  (*From Machine*)
  bI_DeviceOnline            : BOOL;	(*Check link to device*)
  bI_Sensor_pA               : BOOL;	(*Physical sensor feedback for pA Position *)
  bI_Sensor_pB               : BOOL;	(*Physical sensor feedback for pB Position *)
  bI_SystemReady             : BOOL;	(*General ready flag*)
  bI_MovementAllowed         : BOOL;	(*No collision danger*)
  bI_HomingAllowed           : BOOL;	(*Homing allowed*)
  bI_SafetyOk                : BOOL;	(*Safety ok for movement*)
  bI_AbortCleaning           : BOOL;	(*Abort cleaning, drive to pA*)

  (*Commands from Cleaning Process Controller*)
  sI_CleanDevCmd             : ST_CLEANING_DEV_CMD;	(*Initialize operation*)

  (*From User*)
  sI_ManualCommands          : ST_MANUAL_CMD;
  bI_AckFault                : BOOL;	(* Acknowledge errors*)
  bI_Enable                  : BOOL;	(* Enable PrintUnit axis*)
  fI_Position_p1             : REAL;
  fI_Position_p2             : REAL;
  fI_Position_A              : REAL;
  fI_Position_B              : REAL;
  fI_PositionTolerance       : REAL := 0.001;
  fI_SetPositionValue        : REAL := 0.0;    (*Set position value [m]*)
  sI_SpeedDef_Y              : ST_SPEEDS;	(*Speed defs*)
  bI_ShinyMode               : BOOL;	(*Cleaning option*)
  bI_EnableBinClean          : BOOL := TRUE;

  (*From Motor Controller*)
  eI_ELmodule_State          : EN_EL7201_STATE;	(*Feedback from Axis*)
  bI_MoveDone                : BOOL;
  fI_CurrentPosition         : REAL;

  pC_MsgInterface            : POINTER TO ST_ADS_MSG_IF;
  iC_BlockId                 : INT;
END_VAR

VAR_OUTPUT
  (*To Cleaning Head*)
  bO_EnableClnHead           : BOOL;
  bO_EnableVacuum            : BOOL;

  (*To Motor Controller*)
  fO_TargetPosition          : REAL;	(*Target position for axis*)
  fO_SpeedLimit              : REAL;	(*Speed limit for axis*)
  bO_MoveEnable              : BOOL;	(*Move enable for axis*)
  bO_RegActive               : BOOL;	(*Close control loop for axis*)
  bO_FaultReset              : BOOL;	(*Fault reset for axis*)
  bO_SetPosition             : BOOL; (*Reset Encoder*)
  bO_PositionUnknown         : BOOL; (*Position of axis is unknown*)

  (*To machine/user*)
  sO_CleanDevStatus          : ST_CLEANING_DEV_STATUS;	(*Initialize operation*)
  sO_ClnHead_Mvt_Status      : ST_CH_MVT_STATUS;
  bO_CleanAborted            : BOOL;  (*Cleaning aborted*)
END_VAR

VAR
  cL_State                   : BYTE;	(*State type*)
  bL_CleaningActive          : BOOL;
  bL_AfterCleaning           : BOOL := FALSE;
  bL_AxisReady               : BOOL;
  bL_CleanActive             : BOOL;
  bL_MoveAReq                : BOOL;
  bL_MoveBReq                : BOOL;
  bL_MoveDone                : BOOL;
  bL_SafeRunningCondition    : BOOL;
  bL_SafeMoveNeg             : BOOL;
  bL_SafeMovePos             : BOOL;
  bL_Ref_Known               : BOOL := FALSE;
  bL_MoveStarted             : BOOL := FALSE;
  bL_MoveStartRequested      : BOOL := FALSE;

  bL_InPosA                  : BOOL;
  bL_InPosB                  : BOOL;

  wL_ErrorCode               : WORD;

  bL_MotionActive            : BOOL;

  tL_TimerSurv               : TON;			(* Timer for Motorization check *)
  tL_TimerSensor             : TON;			(* Timer for Sensor check *)
  bL_memRefSensor            : BOOL;
  bL_memAck                  : BOOL;
  bL_mem_MotionActive        : BOOL;
  bL_mem_MoveEnable          : BOOL;
  bL_FirstRun                : BOOL := TRUE;
  tL_TonMoveAReq             : TON;			(* Timer for moving back to A *)

  (*Messaging*)
  fB_MsgQueue                : FB_MSG_QUEUE;
  fB_MsgHandler              : FB_MSG_HANDLER;
  sL_MsgConfig               : ST_MSG_CONFIG;
  fB_Msg                     : ARRAY [1..iC_NUM_MSG] OF FB_MESSAGE;
END_VAR

VAR CONSTANT
	(*State*)
  cL_IDLE_A                  : BYTE := 0;										(*Idle-State @ Start*)
  cL_MOVE_P1                 : BYTE := 10;										(*Move to Position where Cleaning starts*)
  cL_ENABLE_CLEAN            : BYTE := 20;										(*Enable Cleaning System*)
  cL_MOVE_P2                 : BYTE := 30;										(*Move to Position where Cleaning stops*)
  cL_DISABLE_CLEAN           : BYTE := 40;										(*Disable Cleaning System*)
  cL_MOVE_A                  : BYTE := 50;										(*Move to start*)
  cL_MOVE_A_CLEANBIN         : BYTE := 51;										(*Move to start with cleaning the bin*)
  cL_MOVE_B                  : BYTE := 60;										(*Move to end*)
  cL_IDLE_B                  : BYTE := 70;										(*Idle-State @ Stop*)
  cL_UNKNOWN                 : BYTE := 80;										(*Position unknown*)

  iC_NUM_MSG                 : INT  := 1;
END_VAR

tL_TimerSurv.PT := T#3s;
tL_TimerSurv();
tL_TimerSensor.PT := T#105s	;	(* 1meter at 10mm*)
tL_TimerSensor();

IF bL_FirstRun THEN
	bL_FirstRun     := FALSE;
	bL_memRefSensor := bI_Sensor_pA;
END_IF;

(*----------------------------------------------------------------------------------------------------------------------------------------------- *)
(*Running Conditions  For Cleaning Head  *)
(*----------------------------------------------------------------------------------------------------------------------------------------------- *)
IF bI_SystemReady AND bI_DeviceOnline AND bI_MovementAllowed AND bI_SafetyOk AND (wL_ErrorCode = 0 OR wL_ErrorCode.5)THEN	(*Dont check limit switch here*)
	bL_SafeRunningCondition := TRUE;
ELSE
	bL_SafeRunningCondition := FALSE;
END_IF;

bL_SafeMoveNeg := bL_SafeRunningCondition AND NOT bI_Sensor_pA AND bI_MovementAllowed;
bL_SafeMovePos := bL_SafeRunningCondition AND NOT bI_Sensor_pB AND bI_MovementAllowed;

IF NOT bI_DeviceOnline THEN
	bL_Ref_Known := FALSE;				(*Reset Reference when link to device is lost, e.g. when machine power off*)
END_IF;

(*----------------------------------------------------------------------------------------------------------------------------------------------- *)
(*Position detection*)
(*----------------------------------------------------------------------------------------------------------------------------------------------- *)

IF     (fI_CurrentPosition >= (fI_Position_A - fI_PositionTolerance)
   AND  fI_CurrentPosition <= (fI_Position_A + fI_PositionTolerance)) OR bI_Sensor_pA
THEN
	bL_InPosA := TRUE;
	bL_InPosB := FALSE;
ELSIF  fI_CurrentPosition >= (fI_Position_B - fI_PositionTolerance)
   AND fI_CurrentPosition <= (fI_Position_B + fI_PositionTolerance)
THEN
	bL_InPosA := FALSE;
	bL_InPosB := TRUE;
ELSE
	bL_InPosA := FALSE;
	bL_InPosB := FALSE;
END_IF;


(*----------------------------------------------------------------------------------------------------------------------------------------------- *)
(* Motion Control For the Cleaning Head 																																																					*)
(*----------------------------------------------------------------------------------------------------------------------------------------------- *)

(*----------------------------------------------------------------------------------------------------------------------------------------------- *)
(*------------------------------------------- Motion Control For the Cleaning Unit   ------------------------------------------------------------ *)
(*----------------------------------------------------------------------------------------------------------------------------------------------- *)
IF NOT bL_Ref_Known THEN	(* if the Y axis hasn't been initialized with Ref Sensor*)
	bL_AxisReady := FALSE;

	IF bI_Sensor_pA AND NOT bL_memRefSensor AND NOT bL_Ref_Known THEN
		bL_Ref_Known    := TRUE;											(* When the sensor is activated, Save the correction value*)
		bL_MotionActive := FALSE;
		bO_SetPosition  := TRUE;											(*Initialize position to preset value*)
		bL_AxisReady    := TRUE;

		fO_TargetPosition := fI_SetPositionValue;
	ELSE
		IF bI_Sensor_pA AND bL_memRefSensor THEN
			fO_TargetPosition := fI_CurrentPosition + 0.01;            (*@@@@CONST, change to JOG_NEGATIVE*)
			fO_SpeedLimit     := sI_SpeedDef_Y.fP_ServiceSpeed;        (* Start backward motion, the motor will run until Ref Sensor is ON*)
			bL_MotionActive   := bI_HomingAllowed;
			bO_SetPosition    := FALSE;
		ELSE
			fO_TargetPosition := -100.0;                               (*@@@@CONST, change to JOG_NEGATIVE*)
			fO_SpeedLimit     := sI_SpeedDef_Y.fP_ServiceSpeed * 0.1;  (* Start backward motion, the motor will run until Ref Sensor is ON*)
			bL_MotionActive   := bI_HomingAllowed;
			bO_SetPosition    := FALSE;
		END_IF;
    (*Security check if sensor malfunction:*)
    (*The CH tries to leave the sensor and drives to side B.*)
    (*If sensor malfunction the axis drives only to the end and stops there.*)
    IF (fO_TargetPosition >= fI_Position_B) THEN
      bL_Ref_Known    := FALSE;
      bL_MotionActive := FALSE;
      bO_SetPosition  := FALSE;
      bL_AxisReady    := FALSE;
		END_IF
	END_IF;
ELSE	(* If the axis has been initialized *)
	IF sI_CleanDevCmd.bService THEN
		ServiceMode();
	ELSE
		ProductionMode();
	END_IF;
END_IF;
bL_memRefSensor := bI_Sensor_pA;				(* Memorization of the Ref sensor state for edge detection*)
bO_RegActive    := bI_Enable AND  bL_SafeRunningCondition;

IF fI_CurrentPosition < fO_TargetPosition THEN			(*  is UP mouvement *)
	bO_MoveEnable := bL_MotionActive AND bL_SafeMovePos;
ELSE																								(*  is DOWN mouvement *)
	bO_MoveEnable := bL_MotionActive AND bL_SafeMoveNeg;
END_IF;

(*----------------------------------------------------------------------------------------------------------------------- *)
(* Output Structure Data Update  																																													*)
(*----------------------------------------------------------------------------------------------------------------------- *)
sO_CleanDevStatus.bBusy     := NOT(bL_AxisReady);
sO_CleanDevStatus.bReady    := bL_AxisReady;
sO_CleanDevStatus.bRefKnown := NOT bO_PositionUnknown;


sO_ClnHead_Mvt_Status.fO_ClnHead_Position := fI_CurrentPosition;
sO_ClnHead_Mvt_Status.bO_Active           := bL_SafeRunningCondition;
sO_ClnHead_Mvt_Status.bO_Ready            := bL_AxisReady;
sO_ClnHead_Mvt_Status.bO_Busy             := bO_MoveEnable;
sO_ClnHead_Mvt_Status.wO_FaultCode        := wL_ErrorCode;

bO_FaultReset := bI_AckFault OR sI_CleanDevCmd.bAckError (*OR fb_MsgQueue.bO_ReceiptMessage*);

IF wL_ErrorCode = 0 THEN
	sO_ClnHead_Mvt_Status.bO_Error := FALSE;
ELSE
	sO_ClnHead_Mvt_Status.bO_Error := TRUE;
END_IF;

(*----------------------------------------------------------------------------------------------------------------------- *)
(*--------------------------------- Fault Diagnosis and Management  ----------------------------------------------------- *)
(*----------------------------------------------------------------------------------------------------------------------- *)
(*Messaging*)
fB_MsgHandler();

IF eI_ELmodule_State = eFault THEN
  fB_Msg[1].bI_Status := TRUE;
ELSE
  fB_Msg[1].bI_Status := FALSE;
END_IF;
fB_Msg[1]();

fB_MsgQueue();


IF (bI_AckFault OR sI_CleanDevCmd.bAckError) AND NOT bL_memAck THEN
	tL_TimerSurv.IN   := FALSE;
	tL_TimerSensor.IN := FALSE;
END_IF;

IF bI_AckFault (*OR fb_MsgQueue.bO_ReceiptMessage*) OR sI_CleanDevCmd.bAckError THEN
	wL_ErrorCode := 0;
END_IF;

IF bI_ClnHeadError THEN	(* Clean Head work status faulty *)
	wL_ErrorCode.1 := TRUE ;
END_IF;

IF (bI_Sensor_pB AND bI_Sensor_pA) THEN			(* Sensor Fault : pB and pA can't be active at the same time *)
	wL_ErrorCode.2 := TRUE ;
END_IF;

IF (sI_SpeedDef_Y.fP_PlaceSpeed=0) OR  (sI_SpeedDef_Y.fP_WorkSpeed=0) OR (sI_SpeedDef_Y.fP_ServiceSpeed=0) THEN	(* Speed Configuration not done *)
	wL_Errorcode.6 := TRUE;
END_IF;

IF (fI_Position_p1=0) OR (fI_Position_p2=0) THEN		(* Position Configuration not done *)
	wL_ErrorCode.7 := TRUE;
END_IF;

IF (eI_ELmodule_State = eFault) OR NOT bI_DeviceOnline THEN
	wL_ErrorCode.8 := TRUE;						(* EL7342 module fault *)
END_IF;

(*IF eI_ELmodule_State=eEstopped THEN
	wL_ErrorCode.15 :=TRUE;						(* EL7342 module fault *)
END_IF;*)

IF wl_ErrorCode = 0 THEN
	sO_CleanDevStatus.bError := FALSE;
ELSE
	sO_CleanDevStatus.bError := TRUE;
END_IF;

bL_mem_MoveEnable   := bO_MoveEnable;
bL_mem_MotionActive := bL_MotionActive;
bL_memAck           := bI_AckFault (*OR fb_MsgQueue.bO_ReceiptMessage*) OR sI_CleanDevCmd.bAckError;

ACTION CleaningProcess:
(*Default*)
bL_MotionActive   := FALSE;
bO_EnableClnHead  := FALSE;
bO_EnableVacuum   := FALSE;
fO_SpeedLimit     := 0;					(*Default speed*)
fO_TargetPosition := fI_Position_A;
bL_MoveDone       := FALSE;
bO_CleanAborted   := FALSE;

(*State Machine -----------------------------------------------------------------*)
CASE cL_State OF
	cL_UNKNOWN:
		IF bL_InPosA THEN	(*The position may be unknown, go automatically to A*)
			bL_MotionActive := FALSE;
			cL_State        := cL_IDLE_A;
			bL_MoveDone     := TRUE;
		ELSE
			IF bL_SafeMovePos OR bL_SafeMoveNeg THEN
				bL_MotionActive := TRUE;
				bL_MoveDone     := FALSE;
			ELSE
				bL_MotionActive := FALSE;
				bL_MoveDone     := TRUE;
			END_IF;
			fO_TargetPosition := fI_Position_A;
			cL_State          := cL_UNKNOWN;
		END_IF;
		fO_SpeedLimit := sI_SpeedDef_Y.fP_PlaceSpeed;
(*		bL_MoveDone:=FALSE;*)

	cL_IDLE_A: 		(*No active operation, the head is at position A*)
		IF bL_InPosA THEN 					(*Position ok*)
			IF bL_MoveBReq THEN					(*Command to move to other end*)
				IF bL_CleanActive THEN		(*When cleaning enabled*)
					cL_State  := cL_MOVE_P1;	(*go step-by-step*)
				ELSE				  							(*otherwise*)
					cL_State  := cL_MOVE_B;		(*go direct*)
				END_IF;
				bL_MoveDone := FALSE;
			ELSE
				bL_MoveDone := TRUE;
			END_IF;
		ELSE	(*Position lost*)
			cL_State    := cL_UNKNOWN;			(*Reinit*)
			bL_MoveDone := FALSE;
		END_IF;

	cL_MOVE_P1: 		(*Move to position P1*)
		IF fI_CurrentPosition < fI_Position_p1 AND NOT (bI_Sensor_pB OR bL_InPosB) THEN
			cL_State        := cL_MOVE_P1;
			bL_MotionActive := TRUE;
    ELSIF bI_AbortCleaning THEN
			cL_State        := cL_MOVE_A;
			bL_MotionActive := FALSE;
      bO_CleanAborted := TRUE;
		ELSE
			cL_State        := cL_ENABLE_CLEAN;
			bL_MotionActive := FALSE;
		END_IF;
		fO_TargetPosition := fI_Position_p1;
		fO_SpeedLimit     := sI_SpeedDef_Y.fP_PlaceSpeed;
		bL_MoveDone       := FALSE;

	cL_ENABLE_CLEAN:	(*Enable Clean Head Valves, Vacuum, etc...*)
		bO_EnableClnHead := TRUE;
		bO_EnableVacuum	 := TRUE;
		IF bI_ClnHeadEnabled THEN
			cL_State        := cL_MOVE_P2;
    ELSIF bI_AbortCleaning THEN
			cL_State        := cL_MOVE_A;
      bO_CleanAborted := TRUE;
		ELSE
			cL_State        := cL_ENABLE_CLEAN;
		END_IF;
		bL_MoveDone       := FALSE;
		bL_AfterCleaning  := TRUE;	(*Set Flag that bin has to be cleaned afterwards*)

	cL_MOVE_P2: 		(*Move to position P2*)
		bO_EnableClnHead  := TRUE;
		bO_EnableVacuum   := TRUE;
		IF fI_CurrentPosition < fI_Position_p2 AND NOT (bI_Sensor_pB OR bL_InPosB) THEN
			cL_State        := cL_MOVE_P2;
			bL_MotionActive := TRUE;
    ELSIF bI_AbortCleaning THEN
			cL_State        := cL_MOVE_A;
			bL_MotionActive := FALSE;
      bO_CleanAborted := TRUE;
		ELSE
			cL_State        := cL_DISABLE_CLEAN;
			bL_MotionActive := FALSE;
		END_IF;
		fO_TargetPosition := fI_Position_p2;
		IF bI_ShinyMode THEN
			fO_SpeedLimit := sI_SpeedDef_Y.fP_WorkSpeed/2;
		ELSE
			fO_SpeedLimit := sI_SpeedDef_Y.fP_WorkSpeed;
		END_IF;
		bL_MoveDone := FALSE;

	cL_DISABLE_CLEAN:	(*Disable Clean Head Valves, Vacuum, etc...*)
		IF NOT bI_ClnHeadEnabled THEN
			cL_State := cL_MOVE_B;
		ELSE
			cL_State := cL_DISABLE_CLEAN;
		END_IF;
		bL_MoveDone := FALSE;

	cL_MOVE_B:	(*Move to position B*)
		IF bL_InPosB THEN
			cL_State        := cL_IDLE_B;
			bL_MotionActive := FALSE;
    ELSIF bI_AbortCleaning THEN
			cL_State        := cL_MOVE_A;
			bL_MotionActive := FALSE;
      bO_CleanAborted := TRUE;
		ELSE
			cL_State        := cL_MOVE_B;
			bL_MotionActive := TRUE;
		END_IF;
		fO_TargetPosition := fI_Position_B;
		fO_SpeedLimit     := sI_SpeedDef_Y.fP_PlaceSpeed;
		bL_MoveDone       := FALSE;
		bO_EnableVacuum   := TRUE;

	cL_IDLE_B: 		(*No active operation, the head is at position B*)
		IF bL_MoveAReq THEN					(*Command to move to other end*)
			IF bL_AfterCleaning AND bI_EnableBinClean AND NOT bI_AbortCleaning THEN
				cL_State := cL_MOVE_A_CLEANBIN;	(*go direct, clean bin*)
			ELSE
				cL_State := cL_MOVE_A;	(*go direct, no cleaning*)
			END_IF;
			bL_MoveDone := FALSE;
		ELSE
			bL_MoveDone := TRUE;
		END_IF;

		IF NOT bL_InPosB THEN 		(*Position lost*)
			;	(*Do nothing*)
		END_IF;

	cL_MOVE_A:
		IF bL_InPosA THEN
			bL_MotionActive := FALSE;
			cL_State        := cL_IDLE_A;
      tL_TonMoveAReq(IN := FALSE);             (*Delay for move back to A*)
		ELSE
      tL_TonMoveAReq(IN := TRUE, PT := T#2S);  (*Delay for move back to A*)
			bL_MotionActive := tL_TonMoveAReq.Q;
			cL_State        := cL_MOVE_A;
		END_IF;
		fO_TargetPosition := fI_Position_A;
		fO_SpeedLimit     := sI_SpeedDef_Y.fP_PlaceSpeed;
		bL_MoveDone       := FALSE;

	cL_MOVE_A_CLEANBIN:
		IF bL_InPosA OR bI_Sensor_pA THEN
			bL_MotionActive := FALSE;
			cL_State        := cL_IDLE_A;
			bL_AfterCleaning:= FALSE;
      tL_TonMoveAReq(IN := FALSE);             (*Delay for move back to A*)
		ELSE
      tL_TonMoveAReq(IN := TRUE, PT := T#2S);  (*Delay for move back to A*)
			bL_MotionActive := tL_TonMoveAReq.Q;
			cL_State        := cL_MOVE_A_CLEANBIN;
			bO_EnableVacuum := bI_EnableBinClean AND NOT bI_AbortCleaning;
		END_IF;
		fO_TargetPosition := fI_Position_A;
		fO_SpeedLimit     := sI_SpeedDef_Y.fP_PlaceSpeed;
		bL_MoveDone       := FALSE;
END_CASE;
END_ACTION

ACTION Init:
	(*Messages*)
	sL_MsgConfig.bI_Enable       := TRUE;
	sL_MsgConfig.pI_FbMsgHandler := ADR(fB_MsgHandler);
	fB_MsgHandler.pI_MsgQueue    := ADR(fB_MsgQueue);
	fB_MsgQueue.pI_MsgInterface  := pC_MsgInterface;
	fB_MsgQueue.cI_MaxElement    := 5;

	fB_Msg[1].iI_MsgLocation     := iC_BlockId;
	fB_Msg[1].pI_MsgConfig       := ADR(sL_MsgConfig);
	fB_Msg[1].iI_MsgNumber       := eCMa_AxisErrorY;
END_ACTION

ACTION ProductionMode:
(*Axis inactive in Production mode*)
bL_MotionActive := FALSE;
bL_AxisReady	  := TRUE;
END_ACTION

ACTION ServiceMode:
(*Mode selection*)
IF sI_CleanDevCmd.bAuto THEN  (*Control by cleaning process*)
  CASE sI_CleanDevCmd.eOperation OF
    eNOP:  (*No operation active*)
      bL_AxisReady        := TRUE;
      bL_CleanActive      := FALSE;
      bL_MoveAReq         := FALSE;
      bL_MoveBReq         := FALSE;
      bO_EnableVacuum     := FALSE;
      bL_MotionActive     := FALSE;
    eOPCLEAN:  (*Cleaning Mode -------------------------------------*)
      IF sI_CleanDevCmd.bInit THEN
        bL_CleanActive    := FALSE;
        bL_AxisReady      := FALSE;
        bL_MoveAReq       := TRUE;
        bL_MoveBReq       := FALSE;

      ELSIF sI_CleanDevCmd.bPrep THEN
        bL_CleanActive    := FALSE;
        bL_AxisReady      := TRUE;
        bL_MoveAReq       := FALSE;
        bL_MoveBReq       := FALSE;

      ELSIF sI_CleanDevCmd.bStart THEN
        bL_CleanActive    := TRUE;
        bL_AxisReady      := FALSE;
        bL_MoveAReq       := FALSE;
        bL_MoveBReq       := TRUE;
      ELSIF sI_CleanDevCmd.bStop THEN
        bL_CleanActive    := FALSE;
        bL_AxisReady      := FALSE;
        bL_MoveAReq       := TRUE;
        bL_MoveBReq       := FALSE;
      ELSE  (*Command removed, wait until axis finished movement*)
        IF bL_MoveDone = FALSE THEN
          bL_AxisReady := FALSE;
          (*Keep other flags as they are*)
        ELSE
          bL_CleanActive  := FALSE;
          bL_AxisReady    := TRUE;
          bL_MoveAReq     := FALSE;
          bL_MoveBReq     := FALSE;
        END_IF;
      END_IF;
      CleaningProcess();        (*Run Cleaning process state machine*)

    eOPCAPENTER:
      IF sI_CleanDevCmd.bInit THEN
        bL_CleanActive    := FALSE;
        bL_AxisReady      := FALSE;
        bL_MoveAReq       := TRUE;
        bL_MoveBReq       := FALSE;

    ELSIF sI_CleanDevCmd.bPrep OR sI_CleanDevCmd.bStart OR sI_CleanDevCmd.bStop THEN
        bL_CleanActive    := FALSE;
        bL_AxisReady      := TRUE;
        bL_MoveAReq       := FALSE;
        bL_MoveBReq       := FALSE;

      ELSE  (*Command removed, wait until axis finished movement*)
        IF bL_MoveDone = FALSE THEN
          bL_AxisReady    := FALSE;
          (*Keep other flags as they are*)
        ELSE
          bL_CleanActive  := FALSE;
          bL_AxisReady    := TRUE;
          bL_MoveAReq     := FALSE;
          bL_MoveBReq     := FALSE;
        END_IF;
      END_IF;
      CleaningProcess();        (*Run Cleaning process state machine*)

    eOPCAPEXIT:
      IF sI_CleanDevCmd.bPrep THEN
        bL_CleanActive    := FALSE;
        bL_AxisReady      := FALSE;
        bL_MoveAReq       := TRUE;
        bL_MoveBReq       := FALSE;

      ELSE  (*Command removed, wait until axis finished movement*)
        IF bL_MoveDone = FALSE THEN
          bL_AxisReady    := FALSE;
          (*Keep other flags as they are*)
        ELSE
          bL_CleanActive  := FALSE;
          bL_AxisReady    := TRUE;
          bL_MoveAReq     := FALSE;
          bL_MoveBReq     := FALSE;
        END_IF;
      END_IF;
      CleaningProcess();        (*Run Cleaning process state machine*)

    eOPPURGE, eOPMAINT, eOPSHUTTEROPEN:  (*Other Mode -------------------------------------*)
      bL_AxisReady    := TRUE;
      bL_CleanActive  := FALSE;
      bL_MotionActive := FALSE;
      bO_EnableVacuum := FALSE;
      bL_MotionActive := FALSE;

  ELSE
    bO_EnableVacuum := FALSE;
    bL_AxisReady    := TRUE;
    bL_CleanActive  := FALSE;
    bL_MotionActive := FALSE;
  END_CASE;

  (*In case of abort set target position to current position and wait for MoveDone flag*)
  IF sI_CleanDevCmd.bAbort THEN
    fO_TargetPosition := fI_CurrentPosition;
    cL_State          := cL_UNKNOWN;  (*Reset cleaning process state machine*)
  END_IF;

ELSE    (* MANUAL MODE *)
  fO_SpeedLimit    := sI_SpeedDef_Y.fP_ServiceSpeed;
  bO_EnableClnHead := FALSE;

  IF sI_ManualCommands.bI_Do = TRUE AND sI_ManualCommands.bI_Undo = FALSE THEN
    fO_TargetPosition := sI_ManualCommands.fI_Start_position;
    bL_AxisReady      := FALSE;
    cL_State := cL_UNKNOWN;  (*Reset cleaning process state machine*)
  ELSIF sI_ManualCommands.bI_Do = FALSE AND sI_ManualCommands.bI_Undo = TRUE THEN
    fO_TargetPosition := sI_ManualCommands.fI_Stop_position;
    bL_AxisReady      := FALSE;
    cL_State := cL_UNKNOWN;  (*Reset cleaning process state machine*)
  ELSE
    fO_TargetPosition := fI_CurrentPosition;
    bL_AxisReady      := TRUE;
  END_IF;
  bL_MotionActive := sI_ManualCommands.bI_Do OR sI_ManualCommands.bI_Undo;
END_IF;
END_ACTION

END_FUNCTION_BLOCK

// ---- POUs/Machine/CleaningStation/FB_CH_PROCESS_CTRL.TcPOU
FUNCTION_BLOCK FB_CH_PROCESS_CTRL
(*************************************************************************************************)
(*  FILENAME:    FB_CH_PROCESS_CTRL                                                              *)
(*  PROJECT:     CALMAR PUPLC                                                                    *)
(*  COPYRIGHT:   All rights reserved (c) Wifag//Polytype, Fribourg/Switzerland (2019)            *)
(*  ENVIRONMENT: TwinCAT PLC                                                                     *)
(*  VERSION:     <version>                                                                       *)
(*************************************************************************************************)
(*  DESCRIPTION:                                                                   <description> *)
(*    This function pilots the Cleaning Head valves.                                             *)
(*    It sends the commands from the FB_CH_MOTION_CTRL to the outputs that controls the valves.  *)
(*                                                                                </description> *)
(*************************************************************************************************)

VAR_INPUT
  (*From Motion Control*)
  bI_EnableClnHead      : BOOL;

  (*From User*)
  bI_WithOutLiquid      : BOOL;
  bI_AckFault           : BOOL;
  tI_VacuumTimer        : TIME := T#2500MS;
  tI_PumpTimer          : TIME := T#1000MS;

  (*From machine*)
  bI_RunningConditions  : BOOL;
  bI_VaccumON           : BOOL;
  bI_NozzleON           : BOOL;
END_VAR

VAR_OUTPUT
  (*To motion control*)
  bO_ClnHeadEnabled     : BOOL;
  bO_ClnHeadError       : BOOL;

  (*To cleaning devices*)
  bO_NozzleActive       : BOOL;
  bO_VaccumActive       : BOOL;
  bO_PumpActive         : BOOL;
END_VAR

VAR
  fb_TonVaccumTimer     : TON;
  fb_TonNozzleTimer     : TON;
  fb_TonTimerSurv       : TON;
  fb_TonPumpTimer       : TON;
  fb_RTrigEnableClnHead : R_TRIG;

  bL_memVaccumCleaning  : BOOL;
  bL_memNozzleCleaning  : BOOL;

  wL_ErrorCode          : WORD;
END_VAR

(* -------------- Timer Settings -------------- *)
fb_TonVaccumTimer.PT := tI_VacuumTimer;
fb_TonNozzleTimer.PT := T#100MS;
fb_TonTimerSurv.PT   := T#2600MS;
IF tI_PumpTimer > fb_TonVaccumTimer.PT THEN
  fb_TonPumpTimer.PT := T#0S;
ELSE
  fb_TonPumpTimer.PT := fb_TonVaccumTimer.PT - tI_PumpTimer;
END_IF

fb_TonVaccumTimer();
fb_TonNozzleTimer();
fb_TonTimerSurv();
fb_TonPumpTimer();

(* ----------------- Rising and Falling Edge Detection for Timer Start --------------- *)
IF bO_VaccumActive <> bL_memVaccumCleaning THEN        (* The timer for Vaccom ON_OFF will start  *)
  fb_TonVaccumTimer.IN := TRUE;                        (* on each edge of the vavle control bit *)
  fb_TonTimerSurv.IN   := TRUE;                        (* start surveillance of the valve *)
END_IF;
(* This timer function is used because *)
(* the system doesn't have a sensor feedback information *)
(* start surveillance of the valve *)

IF bO_NozzleActive <> bL_memNozzleCleaning THEN        (* The timer for Nozzle ON_OFF will start *)
  fb_TonNozzleTimer.IN := TRUE;                        (* on each edge of the valve control bit*)
  fb_TonTimerSurv.IN   := TRUE;                        (* start surveillance of the valve *)
END_IF;

fb_RTrigEnableClnHead(CLK := bI_EnableClnHead);
IF fb_RTrigEnableClnHead.Q THEN
  fb_TonPumpTimer.IN := TRUE;                          (* Timer for cleaner pump *)
END_IF

(* ----------------------- Memorization for Edge Detection ------------------------ *)
bL_memVaccumCleaning := bO_VaccumActive;
bL_memNozzleCleaning := bO_NozzleActive;


(* --------------------- Timer Count Finished --------------------- *)
IF fb_TonVaccumTimer.Q THEN                            (* When the timer for the Vaccum feedback is finished*)
  IF bI_EnableClnHead THEN                             (* Check if the process is for a  Cleaning start*)
    bI_VaccumON := TRUE;                               (* --> Send a sensor ON feedback *)
  ELSE                                                 (* Check if the process is for a Cleaning stop*)
    bI_VaccumON := FALSE;                              (* --> Send a sensor OFF feddback*)
  END_IF;
END_IF;

IF fb_TonNozzleTimer.Q THEN                            (* Same code for the Nozzle *)
  IF bI_EnableClnHead THEN
    bI_NozzleON := TRUE;
  ELSE
    bI_NozzleON := FALSE;
  END_IF;
END_IF;

IF fb_TonPumpTimer.Q THEN
  IF bI_EnableClnHead THEN
    bO_PumpActive := TRUE;
  END_IF;
END_IF;


(* ------------ Valves Controls  -------------- *)
IF bI_RunningConditions AND (wL_ErrorCode = 0) THEN    (* if the running conditions are met and the Cleaning Head is operationnal*)
  IF bI_EnableClnHead THEN                             (* after the start signal has been received, *)
    bO_VaccumActive := TRUE;                           (* Set the Open Vaccum valve control bit, *)

    IF bI_VaccumON THEN                                (* Once the vaccum valve is opened *)
      fb_TonVaccumTimer.IN := FALSE;                   (* Disable the delay timer *)
      fb_TonTimerSurv.IN   := FALSE;                   (* Stop surveillance of the valve *)

      IF NOT bI_WithOutLiquid THEN
        bO_NozzleActive := TRUE;                       (* Set the Open Nozzle Valve control bit *)

        IF bI_NozzleON THEN                            (* Once the nozzle valve is opened *)
          fb_TonNozzleTimer.IN := FALSE;               (* Disable the delay timer *)
          fb_TonTimerSurv.IN   := FALSE;               (* Stop surveillance of the valve *)
        END_IF;
      END_IF;
    END_IF;
  ELSE                                                 (* When the Cleaning is OFF *)
    bO_NozzleActive := FALSE;                          (* First Stop/Close the Nozzle system to stop the liquid flow *)

    IF NOT bI_NozzleON THEN                            (* Once the Nozzle Valve closed *)
      fb_TonNozzleTimer.IN := FALSE;                   (* Disable the timer delay *)
      fb_TonTimerSurv.IN   := FALSE;                   (* Stop surveillance of the valve *)
      bO_VaccumActive      := FALSE;                   (* Once the nozzle is cut off, the system can stop the vaccum *)

      IF NOT bI_VaccumON THEN                          (* Once the Vaccum is stoped*)
        fb_TonVaccumTimer.IN := FALSE;                 (* Disable the timer delay *)
        fb_TonTimerSurv.IN   := FALSE;                 (* Stop surveillance of the valve *)
      END_IF;
    END_IF;

    fb_TonPumpTimer.IN := FALSE;                       (* Disable the pump timer *)
    bO_PumpActive      := FALSE;
  END_IF;
END_IF;


(* ------------------ Error / Warning Definition ---------------------- *)
(* FAULT : Vaccum valve can't open*)
IF (bO_VaccumActive=TRUE  AND fb_TonTimerSurv.Q AND bI_VaccumON=FALSE ) THEN
  wL_ErrorCode.1 := TRUE;
END_IF;
(* FAULT : Vaccum valve can't close*)
IF (bO_VaccumActive=FALSE AND fb_TonTimerSurv.Q AND bI_VaccumON=TRUE  ) THEN
  wL_ErrorCode.2 := TRUE;
END_IF;
(* FAULT : Nozzle valve can't open *)
IF (bO_NozzleActive=TRUE  AND fb_TonTimerSurv.Q AND bI_NozzleON=FALSE ) THEN
  wL_ErrorCode.3 := TRUE;
END_IF;
(* FAULT : Nozzle valve can't close*)
IF (bO_NozzleActive=FALSE AND fb_TonTimerSurv.Q AND bI_NozzleON=TRUE  ) THEN
  wL_ErrorCode.4 := TRUE;
END_IF;

IF (wL_ErrorCode <> 0) OR NOT bI_RunningConditions THEN
  (* the CH have a problem can't operate, need to put everything in safe mode *)
  bO_NozzleActive := FALSE;
  bO_VaccumActive := FALSE;
  bO_PumpActive   := FALSE;

  fb_TonTimerSurv.IN   := FALSE;
  fb_TonNozzleTimer.IN := FALSE;
  fb_TonVaccumTimer.IN := FALSE;
  fb_TonPumpTimer.IN   := FALSE;
END_IF;

IF bI_AckFault THEN
  wL_ErrorCode := 0;
END_IF;

(* ------------------------- Output Value Update ----------------------- *)
bO_ClnHeadEnabled := bI_VaccumON AND bI_NozzleON;
bO_ClnHeadError   := (wL_ErrorCode <> 0);

END_FUNCTION_BLOCK

// ---- POUs/Machine/CleaningStation/FB_CleanDevice.TcPOU
FUNCTION_BLOCK FB_CleanDevice EXTENDS FB_MachineBase IMPLEMENTS I_CleanDevice
(*************************************************************************************************)
(*  FILENAME:    FB_CleanDevice                                                                  *)
(*  PROJECT:     CALMAR PUPLC                                                                    *)
(*  COPYRIGHT:   All rights reserved (c) Polytype AG, Fribourg/Switzerland (2020)                *)
(*  ENVIRONMENT: TwinCAT PLC                                                                     *)
(*  VERSION:     <version>                                                                       *)
(*************************************************************************************************)
(*  DESCRIPTION:                                                                   <description> *)
(*    add description                                                                            *)
(*                                                                                </description> *)
(*************************************************************************************************)

VAR_INPUT
END_VAR

VAR_OUTPUT
END_VAR

VAR
  bL_Busy      : BOOL;  (*The axis is executing the step of a command*)
  bL_AbortReq  : BOOL;  (*Abort requested*)
  bL_Ready     : BOOL;  (*The axis is ready for a new command*)
  bL_Error     : BOOL;  (*The axis has an error*)
  bL_RefKnown  : BOOL;  (*The axis is initialized*)
  sL_CleanMode : EN_Cleaning_OP;
END_VAR

METHOD mAbort : BOOL
//Reset abort only when not in NOP
IF NOT (sL_CleanMode = eNOP) THEN
  bL_AbortReq := TRUE;
END_IF;

mAbort := TRUE;
END_METHOD

METHOD mAckError 
VAR_INPUT
END_VAR
bL_Error := FALSE;
END_METHOD

METHOD mCapping : BOOL
VAR_INPUT
  iI_Step    : INT;
  bI_ExitCap : BOOL;
END_VAR
; //Implement in subclass

//Required feedback:
//busy => Set when step active, reset when step done
//ready => Set when operation done, reset when operation in progress

(*
CASE iI_Step OF
  0: //Init - Check if axis is not activated, restore safety
    bL_Busy := FALSE;

  1: //Move X axis to outside position
    bL_Busy := FALSE;

  2: //Move Z axis to lift position
    bL_Busy := FALSE;

  3: //End - Do nothing, capping process active
    bL_Busy := FALSE;

  ELSE
    bL_Busy := FALSE;		
END_CASE
*)
END_METHOD

METHOD mCleaning : BOOL
VAR_INPUT
  iI_Step : INT;
END_VAR
; //Implement in subclass

//Required feedback:
//busy => Set when step active, reset when step done
//ready => Set when operation done, reset when operation in progress

(*
CASE iI_Step OF
  0: //Init - Check if axis is not activated, restore safety
    bL_Busy := FALSE;

  1: //Move X axis to outside position
    bL_Busy := FALSE;
    
  2: //Move Z axis to lift position
    bL_Busy := FALSE;
    
  3: //Ensure Y axis is at starting position
    bL_Busy := FALSE;
    
  4: //Move Y axis to clean start position
    bL_Busy := FALSE;

  5: //Wait until cleaning equipment ready
    bL_Busy := FALSE;
    
  6: //Cleaning, Y axis move
    bL_Busy := FALSE;
    
  7: //Wait until cleaning equipment ready
    bL_Busy := FALSE;
    
  8: //Move Y axis to end position
    bL_Busy := FALSE;
    
  9: //Move Z axis to lower position
    bL_Busy := FALSE;
  
  10: //Move Y axis back to start 
    bL_Busy := FALSE;

  11: //End
    bL_Busy := FALSE;
  
  ELSE
    bL_Busy := FALSE;    
END_CASE
*)
END_METHOD

METHOD mErrorRecovery : BOOL
VAR_INPUT
    iI_Step : INT;
END_VAR
//Do nothing
bL_Busy := FALSE;
bL_Ready := TRUE;
END_METHOD

METHOD mInit
VAR_INPUT
END_VAR
bL_RefKnown := FALSE;
bL_AbortReq := FALSE;
END_METHOD

METHOD mOperation : BOOL
VAR_INPUT
  iI_Step : INT;
END_VAR
bL_Ready := FALSE;
CASE sL_CleanMode OF
	eOPSTARTUP:
		mStartup(iI_Step);

	eOPCAPENTER:
		mCapping(iI_Step, bI_ExitCap := FALSE);
		
	eOPCAPEXIT:
		mCapping(iI_Step, bI_ExitCap := TRUE);
		
	eOPCLEAN:
		mCleaning(iI_Step);
		
	eOPPREPSERVICE:
		mService(iI_Step);
		
	eOPGOTOPROD:
		mProduction(iI_Step);
    
  eOPEXITERROR:
    mErrorRecovery(iI_Step);
		
	//Add more	
		
	ELSE
		bL_Ready := TRUE;
END_CASE
END_METHOD

METHOD mProduction : BOOL
VAR_INPUT
  iI_Step : INT;
END_VAR
; //Implement in subclass

//Required feedback:
//busy => Set when step active, reset when step done
//ready => Set when operation done, reset when operation in progress

(*
CASE iI_Step OF
  0: //Init - Check if axis is not activated, restore safety
    bL_Busy := FALSE;

  1: //Move Z axis to lower position
    bL_Busy := FALSE;

  2: //Move X axis to inside position
    bL_Busy := FALSE;

  3: //Begin - Do nothing, production active
    bL_Busy := FALSE;

  ELSE
    bL_Busy := FALSE;		
END_CASE
*)
END_METHOD

METHOD mService : BOOL
VAR_INPUT
  iI_Step : INT;
END_VAR
; //Implement in subclass

//Required feedback:
//busy => Set when step active, reset when step done
//ready => Set when operation done, reset when operation in progress

(*
CASE iI_Step OF
  0: //Init - Check if axis is not activated, restore safety
    bL_Busy := FALSE;

  1: //Move X axis to ouside position
    bL_Busy := FALSE;

  2: //Move Z axis to lower position
    bL_Busy := FALSE;

  3: //Begin - Do nothing, service active
    bL_Busy := FALSE;

  4: //End
    bL_Busy := FALSE;

  ELSE
    bL_Busy := FALSE;		
END_CASE
*)
END_METHOD

METHOD mSetMode : BOOL
VAR_INPUT
  sI_CleanMode : EN_CLEANING_OP;
END_VAR
sL_CleanMode := sI_CleanMode;

//Reset abort request as soon as NOP
IF sL_CleanMode = eNOP THEN
  bL_AbortReq := FALSE;
END_IF;


mSetMode := TRUE; //By default all modes supported
END_METHOD

METHOD mStartup : BOOL
VAR_INPUT
  iI_Step : INT;
END_VAR
//Default startup action - do nothing
bL_RefKnown := TRUE;
bL_Busy     := NOT bL_RefKnown;
bL_Ready    := bL_RefKnown;
bL_AbortReq := FALSE;

(*
CASE iI_Step OF
  0: //Init - Check if axis is not activated, restore safety
    bL_Busy := FALSE;

  1: //Move X axis to outside position
    bL_Busy := FALSE;

  2: //Move Z axis to lift position
    bL_Busy := FALSE;

  3: //Begin - Init axis if NOT bL_RefKnown
    bL_Busy := FALSE;

  4: //End
    bL_Busy := FALSE;		

  ELSE
    bL_Busy := FALSE;		
END_CASE
*)
END_METHOD

PROPERTY sStatus : ST_CLEANING_DEV_STATUS
GET
sStatus.bBusy     := bL_Busy;
sStatus.bReady    := bL_Ready; 
sStatus.bError    := bL_Error;
sStatus.bRefKnown := bL_RefKnown;
END_GET
END_PROPERTY

END_FUNCTION_BLOCK

// ---- POUs/Machine/CleaningStation/FB_MachineBase.TcPOU
FUNCTION_BLOCK FB_MachineBase EXTENDS T_NamedBase
(*************************************************************************************************)
(*  FILENAME:    FB_MachineBase                                                                  *)
(*  PROJECT:     CALMAR PUPLC                                                                    *)
(*  COPYRIGHT:   All rights reserved (c) Polytype AG, Fribourg/Switzerland (2020)                *)
(*  ENVIRONMENT: TwinCAT PLC                                                                     *)
(*  VERSION:     <version>                                                                       *)
(*************************************************************************************************)
(*  DESCRIPTION:                                                                   <description> *)
(*    add description                                                                            *)
(*                                                                                </description> *)
(*************************************************************************************************)

VAR_INPUT
	I_MachineStatus : I_MachineStateBase;
END_VAR

END_FUNCTION_BLOCK

// ---- POUs/Machine/CleaningStation/FB_CleaningMotorAxisCH.TcPOU
FUNCTION_BLOCK FB_CleaningMotorAxisCH EXTENDS FB_CleanDevice
VAR_INPUT
  bI_SafeToMove                        : BOOL;
  bI_Emergency                         : BOOL;
  bI_WatchdogError                     : BOOL;
  bI_SafetyOk                          : BOOL;
  bI_UsrAutoMode                       : BOOL;
  bI_UsrService                        : BOOL;
  bI_DevOpActive                       : BOOL;
  bI_CUinPosCappingClean               : BOOL;
  
  //Limit switches
  bI_Sensor_pA                  AT %I* : BOOL;  (*Physical sensor feedback for pA position*)
  bI_Sensor_pB                  AT %I* : BOOL;  (*Physical sensor feedback for pB position*)
  
  //Inputs from EL7201 Terminal
  wI_StatusWord                 AT %I* : UINT; (*Status word: 6041:0*)
  lI_EncoderValue               AT %I* : DINT; (*Encoder value*)
  bI_DeviceOnline               AT %I* : BOOL; (*Check link to device*)
  
  fB_Axis                              : FB_EL7201;    //Axis controller
  
END_VAR

VAR_OUTPUT
  //Outputs to EL7201 Terminal
  wO_ControlWord                AT %Q* : UINT;                         (*Control word:  6040:0*)
  iO_TargetVelocity             AT %Q* : DINT;                         (*Target velocity:  60FF:0*)
END_VAR

VAR
  sADS_CleanAxis                       : FB_ADS_CleanAxis;     //ST_ADS_CLEAN_AXIS;

  //Limit switches
  bL_Sensor_pA                         : BOOL;  (*Negated sensor feedback for pA position*)
  bL_Sensor_pB                         : BOOL;  (*Negated sensor feedback for pB position*)

  fb_TonDeviceOnline                   : TON;
	bIDp_DeviceReset                     : BOOL := FALSE;
	fb_RTrigDeviceReset                  : R_TRIG;

  bL_SafeRunningCondition              : BOOL;
  bL_SafeMoveNeg                       : BOOL;
  bL_SafeMovePos                       : BOOL;
  bL_memRefSensor                      : BOOL;
  bL_FirstRun                          : BOOL := TRUE;

  bL_InPosA                            : BOOL;
  bL_InPosB                            : BOOL;
  
  fb_RFTrigManualMove                  : RF_TRIG;
  sL_CleanDevStatus                    : ST_CLEANING_DEV_STATUS;

  wL_ErrorCode                         : WORD;
  
  (*Messaging*)
  fB_MsgQueue                          : FB_MSG_QUEUE;
  fB_MsgHandler                        : FB_MSG_HANDLER;
  sL_MsgConfig                         : ST_MSG_CONFIG;
  fB_Msg                               : ARRAY [1..iC_NUM_MSG] OF FB_MESSAGE;
END_VAR

VAR PERSISTENT
  fI_Position_p1                       : REAL;           (*[mm]*)
  fI_Position_p2                       : REAL;           (*[mm]*)
  fI_Position_A                        : REAL;           (*[mm]*)
  fI_Position_B                        : REAL;           (*[mm]*)
  fI_PositionTolerance                 : REAL := 0.001;  (*[m]*)
  sI_SpeedDef                          : ST_SPEEDS;  (*Speed defs [mm/s]*)
END_VAR

VAR CONSTANT
  iC_NUM_MSG                           : INT  := 1;
END_VAR

//Limit switches for internal use
bL_Sensor_pA := NOT bI_Sensor_pA;
bL_Sensor_pB := FALSE; (*not existing:  NOT bI_Sensor_pB;*)

(*----------------------------------------------------------------------------------------------------------------------------------------------- *)
(*Running Conditions for Cleaning Head  *)
(*----------------------------------------------------------------------------------------------------------------------------------------------- *)
IF bI_SafeToMove AND I_MachineStatus.pSafetyOk AND I_MachineStatus.pMachineReady AND (wL_ErrorCode = 0 OR wL_ErrorCode.5)THEN  (*Dont check limit switch here*)
  bL_SafeRunningCondition := TRUE;
ELSE
  bL_SafeRunningCondition := FALSE;
END_IF;

bL_SafeMoveNeg := bL_SafeRunningCondition AND NOT bL_Sensor_pA;
bL_SafeMovePos := bL_SafeRunningCondition AND NOT bL_Sensor_pB;

(*Because the WcState sets an error for on cycle, we use this timer to check if the bus is down.*)
fb_TonDeviceOnline(IN := bI_DeviceOnline, PT := T#20MS);
fb_RTrigDeviceReset(CLK := bIDp_DeviceReset);
IF fb_TonDeviceOnline.Q OR fb_RTrigDeviceReset.Q THEN
  bL_RefKnown    := FALSE;        (*Reset Reference when link to device is lost, e.g. when machine power off*)
	wL_ErrorCode.9 := TRUE;
END_IF;

(*----------------------------------------------------------------------------------------------------------------------------------------------- *)
(*Position detection*)
(*----------------------------------------------------------------------------------------------------------------------------------------------- *)
IF     (fB_Axis.fO_ActualPosition >= ((fI_Position_A / 1000) - fI_PositionTolerance)
   AND  fB_Axis.fO_ActualPosition <= ((fI_Position_A / 1000) + fI_PositionTolerance)) OR bL_Sensor_pA
THEN
  bL_InPosA := TRUE;
  bL_InPosB := FALSE;
ELSIF  fB_Axis.fO_ActualPosition >= ((fI_Position_B / 1000) - fI_PositionTolerance)
   AND fB_Axis.fO_ActualPosition <= ((fI_Position_B / 1000) + fI_PositionTolerance)
THEN
  bL_InPosA := FALSE;
  bL_InPosB := TRUE;
ELSE
  bL_InPosA := FALSE;
  bL_InPosB := FALSE;
END_IF;


(*----------------------------------------------------------------------------------------------------------------------------------------------- *)
(* Axis control  *)
(*----------------------------------------------------------------------------------------------------------------------------------------------- *)
fB_Axis.bI_RegActive := bL_SafeRunningCondition AND NOT bL_Error; //Activate controller
fB_Axis.bI_EStop     := I_MachineStatus.pSafetyOk;                //negative logic for bI_EStop

fB_Axis(wI_StatusWord := wI_StatusWord ,lI_EncoderValue := lI_EncoderValue);

fB_Axis.bI_FaultReset := FALSE;

wO_ControlWord    := fB_Axis.wO_ControlWord;
iO_TargetVelocity := fB_Axis.iO_TargetVelocity;


(*----------------------------------------------------------------------------------------------------------------------------------------------- *)
(*Manuell move in hand mode (NOT bI_UsrAutoMode)*)
(*----------------------------------------------------------------------------------------------------------------------------------------------- *)
fb_RFTrigManualMove(CLK := sADS_CleanAxis.bI_ManualMove);
IF     NOT bI_UsrAutoMode 
   AND bI_UsrService
   AND bI_SafetyOk
   AND NOT bI_WatchdogError
   AND bI_CUinPosCappingClean
THEN
  sADS_CleanAxis.setFeedback( bManualMoveCanEx := TRUE
                            , bManualMovekExec := sADS_CleanAxis.bO_ManualMovekExec        // do not change
                            , fAxisPositionVal := sADS_CleanAxis.sO_AxisPosition.fO_Val    // do not change
                            , wErrorCode       := sADS_CleanAxis.wO_ErrorCode              // do not change
                            , bBusy            := sADS_CleanAxis.bO_Busy                   // do not change
                            , bReady           := sADS_CleanAxis.bO_Ready                  // do not change
                            , bError           := sADS_CleanAxis.bO_Error                  // do not change
                            );

  IF sADS_CleanAxis.bI_ManualMove OR fb_RFTrigManualMove.FT THEN
    mManuellMove( bI_Do                  := sADS_CleanAxis.bI_ManualMove
                , fI_TargetPosition      := SEL( sADS_CleanAxis.bI_ManualMove
                                               , (fB_Axis.fO_ActualPosition * 1000)
                                               , sADS_CleanAxis.fI_ManualTargetPos)
                , fL_ManualMoveTolerance := fB_Axis.fI_Tolerance);
  END_IF
ELSE
  sADS_CleanAxis.setFeedback( bManualMoveCanEx := FALSE
                            , bManualMovekExec := sADS_CleanAxis.bO_ManualMovekExec        // do not change
                            , fAxisPositionVal := sADS_CleanAxis.sO_AxisPosition.fO_Val    // do not change
                            , wErrorCode       := sADS_CleanAxis.wO_ErrorCode              // do not change
                            , bBusy            := sADS_CleanAxis.bO_Busy                   // do not change
                            , bReady           := sADS_CleanAxis.bO_Ready                  // do not change
                            , bError           := sADS_CleanAxis.bO_Error                  // do not change
                            );
  sADS_CleanAxis.ResetCommands();

  IF fb_RFTrigManualMove.FT THEN
    mManuellMove( bI_Do                  := FALSE
                , fI_TargetPosition      := (fB_Axis.fO_ActualPosition * 1000)
                , fL_ManualMoveTolerance := fB_Axis.fI_Tolerance);
  END_IF
END_IF
(*Rest command if move is done*)
IF bL_Ready OR bL_Error THEN
  sADS_CleanAxis.ResetCommands();
END_IF

sL_CleanDevStatus := sStatus;

(*ADS Feedback*)
sADS_CleanAxis.setFeedback( bManualMoveCanEx := sADS_CleanAxis.bO_ManualMoveCanEx        // do not change
                          , bManualMovekExec := sADS_CleanAxis.bO_ManualMovekExec        // do not change
                          , fAxisPositionVal := fB_Axis.fO_ActualPosition * 1000
                          , wErrorCode       := wL_ErrorCode
                          , bBusy            := sL_CleanDevStatus.bBusy
                          , bReady           := sL_CleanDevStatus.bReady
                          , bError           := sL_CleanDevStatus.bError
                          );


(*----------------------------------------------------------------------------------------------------------------------------------------------- *)
(* Supervision  *)
(*----------------------------------------------------------------------------------------------------------------------------------------------- *)
(*
TODO: Supervisor
tL_TimerSurv.PT := T#3S;
tL_TimerSurv();
tL_TimerSensor.PT := T#105s  ;  (* 1meter at 10mm*)
tL_TimerSensor();*)

IF bL_FirstRun THEN
  bL_FirstRun     := FALSE;
  bL_memRefSensor := bL_Sensor_pA;
END_IF;

(*----------------------------------------------------------------------------------------------------------------------- *)
(*--------------------------------- Fault Diagnosis and Management  ----------------------------------------------------- *)
(*----------------------------------------------------------------------------------------------------------------------- *)
mErrorHandling();

(*----------------------------------------------------------------------------------------------------------------------- *)
(* Messaging                                                                                                              *)
(*----------------------------------------------------------------------------------------------------------------------- *)
fB_MsgHandler();
fB_Msg[1](bI_Status := bL_Error);
fB_MsgQueue();

METHOD mAckError 
VAR_INPUT
END_VAR
wL_ErrorCode := 0;
mErrorHandling();
fB_Axis.bI_FaultReset := TRUE;
END_METHOD

METHOD mCapping : BOOL
VAR_INPUT
  iI_Step    : INT;
  bI_ExitCap : BOOL;
END_VAR
//Abort: Stop whereever axis is and return
IF bL_AbortReq THEN
  fB_Axis.bI_MoveEnable := FALSE;
  bL_Busy  := FALSE;
  bL_Ready := TRUE;

  RETURN;
END_IF

//Normal operation
bL_Ready := FALSE;
CASE iI_Step OF
	0: //Init - Check if axis is not activated, restore safety
    fB_Axis.bI_MoveEnable := FALSE;
		bL_Busy := FALSE;

  1: //Wait for PU axis to lift
    fB_Axis.bI_MoveEnable   := FALSE;
    bL_Busy                 := FALSE;
    
  2: //Wait for CU axis to move in
    fB_Axis.bI_MoveEnable   := FALSE;
    bL_Busy                 := FALSE;
    
  3: //Move CH to park positiom 
    fB_Axis.fI_TargetPosition := (fI_Position_A / 1000);
    fB_Axis.fI_SpeedLimit     := sI_SpeedDef.fP_PlaceSpeed / 1000;
    
    IF bL_InPosA THEN //Target reached
      fB_Axis.bI_MoveEnable := FALSE;
      bL_Busy               := FALSE;
      bL_Ready              := TRUE;  //Operation complete
    ELSE
      fB_Axis.bI_MoveEnable := bL_SafeMoveNeg;
      bL_Busy               := TRUE;
    END_IF

  4: //Wait for PU axis to lower
    fB_Axis.bI_MoveEnable   := FALSE;
    bL_Busy                 := FALSE;
    
	5: //End - Do nothing, capping process active
    mAckError();
		bL_Busy  := FALSE;
    bL_Ready := TRUE;  //Operation complete

	ELSE
		bL_Busy  := FALSE;		
    bL_Ready := TRUE;  //Operation complete
END_CASE
END_METHOD

METHOD mCleaning : BOOL
VAR_INPUT
  iI_Step : INT;
END_VAR
//Abort: Stop whereever axis is and return
IF bL_AbortReq THEN
  bL_Busy:=FALSE;
  fB_Axis.bI_MoveEnable:=FALSE;
  bL_Ready := TRUE;
  RETURN;
END_IF

//Normal operation
bL_Ready := FALSE;
CASE iI_Step OF
  0: //Init - Check if axis is not activated, restore safety
    bL_Busy := FALSE;

  1: //Wait for PU axis to lift
    fB_Axis.bI_MoveEnable   := FALSE;
    bL_Busy                 := FALSE;
    
  2: //Wait for CU axis to move in
    fB_Axis.bI_MoveEnable   := FALSE;
    bL_Busy                 := FALSE;
    
  3: //Wait for PU axis to lower
    fB_Axis.bI_MoveEnable   := FALSE;
    bL_Busy                 := FALSE;
    
  4: //Ensure CH axis is at starting position
    mAckError();
    fB_Axis.fI_TargetPosition := (fI_Position_A / 1000);
    fB_Axis.fI_SpeedLimit     := sI_SpeedDef.fP_PlaceSpeed / 1000;
    
    IF bL_InPosA THEN
      fB_Axis.bI_MoveEnable := FALSE;
      bL_Busy               := FALSE;
      bL_Ready              := TRUE;  //Operation complete
    ELSE
      fB_Axis.bI_MoveEnable := TRUE;
      bL_Busy               := TRUE;
    END_IF
    
  5: //Move CH to clean start position
    fB_Axis.fI_TargetPosition := (fI_Position_p1 / 1000);
    fB_Axis.fI_SpeedLimit     := sI_SpeedDef.fP_PlaceSpeed / 1000;
    
    IF bL_Sensor_pB OR bL_InPosB THEN //Error
      ; //TODO
    ELSIF fB_Axis.fO_ActualPosition >= (fI_Position_p1 / 1000) THEN //Target reached
      fB_Axis.bI_MoveEnable := FALSE;
      bL_Busy               := FALSE;
      bL_Ready              := TRUE;  //Operation complete
    ELSE
      fB_Axis.bI_MoveEnable := bL_SafeMovePos;
      bL_Busy               := TRUE;
    END_IF

  6: //Wait until cleaning equipment ready
    fB_Axis.bI_MoveEnable   := FALSE;
    bL_Busy                 := FALSE;
    
  7: //Cleaning
    fB_Axis.fI_TargetPosition := (fI_Position_p2 / 1000);
    fB_Axis.fI_SpeedLimit     := sI_SpeedDef.fP_WorkSpeed / 1000;
    
    IF bL_Sensor_pB OR bL_InPosB THEN //Error
      ; //TODO
    ELSIF fB_Axis.fO_ActualPosition >= (fI_Position_p2 / 1000) THEN //Target reached
      fB_Axis.bI_MoveEnable := FALSE;
      bL_Busy               := FALSE;
      bL_Ready              := TRUE;  //Operation complete
    ELSE
      fB_Axis.bI_MoveEnable := bL_SafeMovePos;
      bL_Busy               := TRUE;
    END_IF
    
  8: //Wait until cleaning equipment ready
    fB_Axis.bI_MoveEnable   := FALSE;
    bL_Busy                 := FALSE;
    
  9: //Move CH to end position
    fB_Axis.fI_TargetPosition := (fI_Position_B / 1000);
    fB_Axis.fI_SpeedLimit     := sI_SpeedDef.fP_PlaceSpeed / 1000;
    
    IF bL_InPosB THEN //Target reached
      fB_Axis.bI_MoveEnable := FALSE;
      bL_Busy               := FALSE;
      bL_Ready              := TRUE;  //Operation complete
    ELSE
      fB_Axis.bI_MoveEnable := bL_SafeMovePos;
      bL_Busy               := TRUE;
    END_IF
    
  10: //Wait for PU axis to lift
    fB_Axis.bI_MoveEnable := FALSE;
    bL_Busy               := FALSE;  
  
  11: //Move CH back to start 
    fB_Axis.fI_TargetPosition := (fI_Position_A / 1000);
    fB_Axis.fI_SpeedLimit     := sI_SpeedDef.fP_PlaceSpeed / 1000;
    
    IF bL_InPosA THEN //Target reached
      fB_Axis.bI_MoveEnable := FALSE;
      bL_Busy               := FALSE;
      bL_Ready              := TRUE;  //Operation complete
    ELSE
      fB_Axis.bI_MoveEnable := bL_SafeMoveNeg;
      bL_Busy               := TRUE;
    END_IF

  12: //Wait for PU axis to lower
    fB_Axis.bI_MoveEnable   := FALSE;
    bL_Busy                 := FALSE;
    
  13: //End
    fB_Axis.bI_MoveEnable := FALSE;
    bL_Busy               := FALSE;  
    bL_Ready              := TRUE;  //Operation complete

  ELSE
    bL_Busy  := FALSE;    
    bL_Ready := TRUE;  //Operation complete
END_CASE
END_METHOD

METHOD PRIVATE mErrorHandling
VAR_INPUT
END_VAR
fB_Msg[1].bI_Status := FALSE;

IF (bL_Sensor_pB AND bL_Sensor_pA) THEN			(* Sensor Fault : pB and pA can't be active at the same time *)
	wL_ErrorCode.2 := TRUE ;
END_IF;

IF (sI_SpeedDef.fP_PlaceSpeed=0) OR  (sI_SpeedDef.fP_WorkSpeed=0) OR (sI_SpeedDef.fP_ServiceSpeed=0) THEN	(* Speed Configuration not done *)
	wL_Errorcode.6 := TRUE;
END_IF;

IF (fI_Position_p1=0) OR (fI_Position_p2=0) THEN		(* Position Configuration not done *)
	wL_ErrorCode.7 := TRUE;
END_IF;

IF fB_Axis.eO_EL7201Status = eFault  THEN
	wL_ErrorCode.8 := TRUE;						(* EL7342 module fault *)
	fB_Msg[1].bI_Status := TRUE;
END_IF;


IF wl_ErrorCode = 0 THEN
	bL_Error := FALSE;
ELSE
	bL_Error := TRUE;
END_IF;
END_METHOD

METHOD mErrorRecovery : BOOL
VAR_INPUT
    iI_Step : INT;
END_VAR
//Do nothing
bL_Busy := FALSE;
bL_Ready := TRUE;
END_METHOD

METHOD mInit
VAR_INPUT
END_VAR
	(*Messages*)
	sL_MsgConfig.bI_Enable       := TRUE;
	sL_MsgConfig.pI_FbMsgHandler := ADR(fB_MsgHandler);
	fB_MsgHandler.pI_MsgQueue    := ADR(fB_MsgQueue);
	fB_MsgQueue.pI_MsgInterface  := ADR(sADS_CleanAxis.sO_Message);
	fB_MsgQueue.cI_MaxElement    := 5;

	fB_Msg[1].iI_MsgLocation     := TO_INT(eMa_BLK_CLEANAXIS);
	fB_Msg[1].pI_MsgConfig       := ADR(sL_MsgConfig);
	fB_Msg[1].iI_MsgNumber       := eCMa_AxisErrorY;
END_METHOD

METHOD mManuellMove : BOOL
VAR_INPUT
  bI_Do                  : BOOL;
  fI_TargetPosition      : REAL;
  fL_ManualMoveTolerance : REAL;
END_VAR
fB_Axis.fI_SpeedLimit     := sI_SpeedDef.fP_ServiceSpeed / 1000;
fB_Axis.fI_TargetPosition := fI_TargetPosition / 1000;
IF fB_Axis.fI_TargetPosition > fB_Axis.fO_ActualPosition THEN
  fB_Axis.bI_MoveEnable   := bI_Do AND bL_SafeMovePos;
ELSIF fB_Axis.fI_TargetPosition < fB_Axis.fO_ActualPosition THEN
  fB_Axis.bI_MoveEnable   := bI_Do AND bL_SafeMoveNeg;
ELSE
  fB_Axis.bI_MoveEnable   := bI_Do;
END_IF

bL_Busy  := ABS(fB_Axis.fI_TargetPosition - fB_Axis.fO_ActualPosition) > fL_ManualMoveTolerance;
bL_Ready := NOT (ABS(fB_Axis.fI_TargetPosition - fB_Axis.fO_ActualPosition) > fL_ManualMoveTolerance);  //Operation complete
END_METHOD

METHOD mProduction : BOOL
VAR_INPUT
  iI_Step : INT;
END_VAR
//Nothing to do
fB_Axis.bI_MoveEnable := FALSE;
bL_Busy  := FALSE;
bL_Ready := TRUE;
END_METHOD

METHOD mService : BOOL
VAR_INPUT
  iI_Step : INT;
END_VAR
//Nothing to do
fB_Axis.bI_MoveEnable := FALSE;
bL_Busy  := FALSE;
bL_Ready := TRUE;
END_METHOD

METHOD mStartup : BOOL
VAR_INPUT
  iI_Step : INT;
END_VAR
CASE iI_Step OF
	0: //Init - Check if axis is not activated, restore safety
		bL_Busy := FALSE;

	1,2: //Wait until other axes in place
		bL_Busy := FALSE;

	3: //Begin - Init CH axis if NOT bL_RefKnown
    bL_Busy  := NOT bL_RefKnown;
    bL_Ready := bL_RefKnown;
    
    fB_Axis.bI_SetPosition := bL_RefKnown;
    
    IF NOT bL_RefKnown THEN  (* if the Y axis hasn't been initialized with Ref Sensor*)
      IF bL_Sensor_pA AND NOT bL_memRefSensor AND NOT bL_RefKnown THEN
        bL_RefKnown             := TRUE;                      (* When the sensor is activated, Save the correction value*)
        fB_Axis.bI_SetPosition  := TRUE;                      (*Initialize position to preset value*)
        fB_Axis.bI_MoveEnable   := FALSE;
        bL_Ready                := TRUE;
      ELSE
        IF bL_Sensor_pA AND bL_memRefSensor THEN
          fB_Axis.fI_TargetPosition := fB_Axis.fO_ActualPosition + 0.01;  (*@@@@CONST, change to JOG_NEGATIVE*)
          fB_Axis.fI_SpeedLimit     := sI_SpeedDef.fP_ServiceSpeed / 1000;     (* Start backward motion, the motor will run until Ref Sensor is ON*)
          fB_Axis.bI_MoveEnable     := bL_SafeMovePos;
        ELSIF bL_Sensor_pB THEN (*Security check if sensor malfunction:*)
          ; //Error
        ELSE
          fB_Axis.fI_TargetPosition := -100.0;                               (*@@@@CONST, change to JOG_NEGATIVE*)
          fB_Axis.fI_SpeedLimit     := (sI_SpeedDef.fP_ServiceSpeed * 0.1) / 1000;  (* Start backward motion, the motor will run until Ref Sensor is ON*)
          fB_Axis.bI_MoveEnable     := bL_SafeMoveNeg;
        END_IF;
      END_IF;
    END_IF;

    bL_memRefSensor := bL_Sensor_pA;				(* Memorization of the Ref sensor state for edge detection*)

	4: //End
		bL_Busy  := FALSE;		
    bL_Ready := TRUE;  //Operation complete

	ELSE
		bL_Busy  := FALSE;		
    bL_Ready := TRUE;  //Operation complete
END_CASE
END_METHOD

{attribute 'monitoring' := 'call'}
PROPERTY pInPosA : bool
GET
pInPosA := bL_InPosA;
END_GET
END_PROPERTY

{attribute 'monitoring' := 'call'}
PROPERTY pInPosB : bool
GET
pInPosB := bL_InPosB;
END_GET
END_PROPERTY

END_FUNCTION_BLOCK

// ---- POUs/Machine/CleaningStation/FB_EL7201.TcPOU
FUNCTION_BLOCK FB_EL7201
(*************************************************************************************************)
(*  FILENAME:    FB_EL7201                                                                       *)
(*  PROJECT:     CALMAR PUPLC                                                                    *)
(*  COPYRIGHT:   All rights reserved (c) Wifag//Polytype, Fribourg/Switzerland (2020)            *)
(*  ENVIRONMENT: TwinCAT PLC                                                                     *)
(*  VERSION:     <version>                                                                       *)
(*************************************************************************************************)
(*  DESCRIPTION:                                                                   <description> *)
(*    This function transfers the movement commands to the motor.                                *)
(*                                                                                </description> *)
(*************************************************************************************************)

{library PUBLIC}
VAR_INPUT
  fI_TargetPosition              : REAL;                         (*Target position*)
  fI_Tolerance                   : REAL := 0.0001;               (*Position tolerance*)
  fI_SpeedLimit                  : REAL;                         (*Speed limit*)
  bI_MoveEnable                  : BOOL;                         (*Enable movement*)
  bI_RegActive                   : BOOL;                         (*Regulation active*)
  bI_FaultReset                  : BOOL;                         (*Fault reset*)
  bI_EStop                       : BOOL;                         (*Emergency stop*)
  bI_SetPosition                 : BOOL;                         (*Set position*)

  wI_StatusWord                  : UINT;                         (*Status word: 6041:0*)
  lI_EncoderValue                : DINT;                         (*Encoder value*)
  fI_PosControllerGain           : REAL := 5.0;                  (*Position controller gain*)
  fI_EncoderScaling              : REAL := 1048576;              (*Encoder scaling [counts/rev]*)
  fI_Axis_Scaling                : REAL := 0.010 * 1/10;         (*Axis scaling [m/rev]*)
  fI_SetPositionValue            : REAL := -0.001;               (*Set position value [m]*)
  fI_SpeedScaling                : REAL := 268435;               (*Speed scaling [counts/rev]*)
END_VAR

VAR_OUTPUT
  wO_ControlWord                 : UINT;                         (*Control word:  6040:0*)
  iO_TargetVelocity              : DINT;                         (*Target velocity:  60FF:0*)
  fO_ActualPosition              : REAL;                         (*Actual position [m]*)
  bO_MoveOk                      : BOOL;                         (*Movement ok*)
  eO_EL7201Status                : EN_EL7201_STATE;              (*EL7201 status*)
END_VAR

{library private}
VAR
  fL_Delta_P                     : REAL;                         (*Delta position*)
  fL_CommandSignal               : REAL;                         (*Command signal*)

  tL_TimerRampUP                 : TON;                          (*Timer ramp up*)
  fL_PercentageRampUP            : REAL;                         (*Percentage ramp up*)
  tL_TimerRampDN                 : TON;                          (*Timer ramp down*)
  fL_PercentageRampDN            : REAL;                         (*Percentage ramp down*)

  wL_MaskedStatusWord            : WORD;                         (*Masked status word*)
  bL_memMoveEnable               : BOOL;                         (*Memory enable movement*)
  bL_memSetPosition              : BOOL;                         (*Memory set position*)
  fL_memTargetPosition           : REAL := 0.0;                  (*Memory target position*)
  bL_StopRamp                    : BOOL;                         (*Stop ramp*)
  bL_FirstRun                    : BOOL := TRUE;                 (*First run*)

  fL_Divider                     : REAL;                         (*Divider for percent calculation*)
END_VAR

VAR PERSISTENT
  fL_OffsetEncoder               : DINT;                         (*Offset encoder*)
END_VAR

//Read inputs
Input();

tL_TimerRampUP.PT := T#300MS;
tL_TimerRampUP();

tL_TimerRampDN.PT := T#300MS;
tL_TimerRampDN();

IF NOT bI_MoveEnable AND bL_memMoveEnable THEN
	bL_StopRamp := TRUE;
END_IF;

IF bI_MoveEnable AND NOT bL_memMoveEnable THEN
	fL_memTargetPosition := fI_TargetPosition;
	bO_MoveOK := FALSE;
ELSIF bL_FirstRun THEN
	fL_memTargetPosition := fO_ActualPosition;
END_IF;


IF tL_TimerRampDN.Q THEN
	bL_StopRamp := FALSE;
END_IF;

tL_TimerRampDN.IN := bL_StopRamp;

fL_Divider := TIME_TO_REAL(tL_TimerRampDN.PT);
IF fL_Divider <> 0 THEN
	fL_PercentageRampDN := TIME_TO_REAL(tL_TimerRampDN.ET)/fL_Divider;
END_IF;

tL_TimerRampUP.IN := bI_MoveEnable AND bI_RegActive;

fL_Divider := TIME_TO_REAL(tL_TimerRampUP.PT);
IF fL_Divider <> 0 THEN
	fL_PercentageRampUP := TIME_TO_REAL(tL_TimerRampUP.ET)/fL_Divider;
END_IF;

(* ---------------------- Calculation of the Error Signal between the Target and the Actual Position -----------------*)
fL_Delta_P := fI_TargetPosition - fO_ActualPosition;

(* --------------------------------- Calculation of the Command Signal for the Target Velocity  ---------------------------*)
fL_CommandSignal := fL_Delta_P * fI_PosControllerGain;

(* ----------------------------- Limitation of the Command Signal between +/- SpeedLimit --------------------------------*)
IF fL_CommandSignal > (fI_SpeedLimit) THEN
	fL_CommandSignal:= fI_SpeedLimit;
ELSIF fL_CommandSignal < (-fI_SpeedLimit) THEN
	fL_CommandSignal:=-fI_SpeedLimit;
END_IF;

IF bI_MoveEnable THEN
	IF fI_Axis_Scaling <> 0 THEN
		iO_TargetVelocity:= FC_REAL_TO_DINT((fI_SpeedScaling / fI_Axis_Scaling * fL_CommandSignal * fL_PercentageRampUP));			(* Send the Target velocity command to module *)
	END_IF;
ELSE
	IF fI_Axis_Scaling <> 0 THEN
		iO_TargetVelocity:= FC_REAL_TO_DINT((fI_SpeedScaling / fI_Axis_Scaling * fL_CommandSignal * (1-fL_PercentageRampDN)));	(* Send the Target velocity command to module *)
	END_IF;
END_IF;

(* ---------------------- MDP StateMachine ----------------- *)
MDP_StateMachine();

(* ---------------------- Encoder Offset Calibration ----------------- *)

IF bI_SetPosition AND NOT bL_memSetPosition AND NOT bI_MoveEnable THEN
	IF fI_Axis_Scaling <> 0 THEN
		fL_OffsetEncoder := FC_REAL_TO_DINT((fI_SetPositionValue * fI_EncoderScaling / fI_Axis_Scaling - DINT_TO_REAL(lI_EncoderValue)));
	END_IF;

	fL_memTargetPosition := fO_ActualPosition;
END_IF;

(* ---------------------- Memory ----------------- *)
bL_memSetPosition := bI_SetPosition;
bL_memMoveEnable  := bI_MoveEnable;
bL_FirstRun       := FALSE;

(********************************* END OF FB *****************************************************)

METHOD PRIVATE Input
VAR_INPUT
END_VAR
(*EL7201 Standard: 20 Singleturn bits and 12 Multiturn bits*)
IF (fI_EncoderScaling <> 0) THEN
	fO_ActualPosition := (DINT_TO_REAL(lI_EncoderValue) + DINT_TO_REAL(fL_OffsetEncoder)) * fI_Axis_Scaling / fI_EncoderScaling;
END_IF;

(*Movement done?*)
IF bI_MoveEnable THEN
	IF ABS(fL_memTargetPosition - fO_ActualPosition) < fI_Tolerance*0.2 THEN
		bO_MoveOK := TRUE;
	ELSE
		bO_MoveOK := FALSE;
	END_IF;
ELSE
	IF ABS(fL_memTargetPosition - fO_ActualPosition) < fI_Tolerance THEN
		bO_MoveOK := TRUE;
	ELSE
		bO_MoveOK := FALSE;
	END_IF;
END_IF;
END_METHOD

METHOD PRIVATE MDP_StateMachine
VAR_INPUT
END_VAR
wL_MaskedStatusWord := UINT_TO_WORD(wI_StatusWord) AND 16#006F;

IF NOT bI_EStop THEN
  iO_TargetVelocity := 0;
  eO_EL7201Status   := eEstopped;
  wO_ControlWord    := 16#0000;
  wO_ControlWord    := 16#0002;
ELSE

  CASE wL_MaskedStatusWord OF
      16#0000, 16#0020:            (* ------------------ State : Not Ready to Switch On : x0xx0000 ---------------------- *)
        eO_EL7201Status := eNotReadyToSwitchON ;

      16#0040, 16#0060:            (* ------------------ State : Switch ON Disable : x1xx0000 ---------------------- *)
        eO_EL7201Status := eSwitchONDisabled ;
        wO_ControlWord := 16#0006;

      16#0021:                     (* ------------------ State : Ready To Switch ON : x01x0001---------------------- *)
        eO_EL7201Status := eReadyToSwitchON ;
        IF bI_RegActive=TRUE THEN
          wO_ControlWord := 16#0007;
        END_IF;

      16#0023:                     (* ---------------- State : Switched ON : x01x0011------------------ *)
        eO_EL7201Status := eSwitchedON ;
        IF bI_MoveEnable=TRUE THEN
          wO_ControlWord := 16#000F;
        END_IF;

        IF bI_RegActive=FALSE THEN
          wO_ControlWord := 16#0006;
        END_IF;

      16#0027:                     (* -------------- State : Enabled : x01x0111------------------ *)
        eO_EL7201Status := eEnabled;
        IF (bI_MoveEnable=FALSE AND tL_TimerRampDN.Q) THEN
          wO_ControlWord := 16#0007;
        END_IF;

      16#000F, 16#002F:            (* -------------- State : Fault Reaction Active : x0xx1111----------------- *)
        eO_EL7201Status := eFaultReactionActive ;

      16#0008, 16#0028, 16#0068:   (* --------------- State :  Fault : x0xx1000 ------------------- *)
        eO_EL7201Status := eFault;
        IF bI_FaultReset THEN
          wO_ControlWord := 16#0080;
        ELSE
          wO_ControlWord := 16#0000;
        END_IF;
  END_CASE;
END_IF;
END_METHOD

END_FUNCTION_BLOCK

// ---- POUs/Machine/CleaningStation/FB_CleaningMotorAxisCU.TcPOU
FUNCTION_BLOCK FB_CleaningMotorAxisCU EXTENDS FB_CleanDevice
VAR_INPUT
  bI_SafeToMove                        : BOOL;
  bI_Emergency                         : BOOL;
  bI_WatchdogError                     : BOOL;
  bI_SafetyOk                          : BOOL;
  bI_MachineReady                      : BOOL;
  bI_UsrAutoMode                       : BOOL;
  bI_UsrService                        : BOOL;
  bI_DevOpActive                       : BOOL;
  bI_PUinPosService                    : BOOL;
  
  //Limit switches
  bI_ReferenceSensor            AT %I* : BOOL;  (*Physical sensor feedback reference position*)
  
  //Inputs from EL7201 Terminal
  wI_StatusWord                 AT %I* : UINT; (*Status word: 6041:0*)
  lI_EncoderValue               AT %I* : DINT; (*Encoder value*)
  bI_DeviceOnline               AT %I* : BOOL; (*Check link to device*)
  
  fB_Axis                              : FB_EL7201;    //Axis controller
END_VAR

VAR_OUTPUT
  //Outputs to EL7201 Terminal
  wO_ControlWord                AT %Q* : UINT;                         (*Control word:  6040:0*)
  iO_TargetVelocity             AT %Q* : DINT;                         (*Target velocity:  60FF:0*)
END_VAR

VAR
  sADS_CleanAxis                       : FB_ADS_CleanAxis;     //ST_ADS_CLEAN_AXIS;

  //Limit switches
  bL_ReferenceSensor                   : BOOL;  (*Negated sensor feedback reference position*)

  fb_TonDeviceOnline                   : TON;
	bIDp_DeviceReset                     : BOOL := FALSE;
	fb_RTrigDeviceReset                  : R_TRIG;

  bL_SafeRunningCondition              : BOOL;
  bL_SafeMoveNeg                       : BOOL;
  bL_SafeMovePos                       : BOOL;
  bL_memRefSensor                      : BOOL;
  bL_FirstRun                          : BOOL := TRUE;

  fL_ManualMoveTolerance               : REAL := 0.001;
  fb_RFTrigManualMove                  : RF_TRIG;
  sL_CleanDevStatus                    : ST_CLEANING_DEV_STATUS;
  
  bL_InPosCappClean                    : BOOL;
  bL_InPosPark                         : BOOL;
  
  wL_ErrorCode                         : WORD;
  
  (*Messaging*)
  fB_MsgQueue                          : FB_MSG_QUEUE;
  fB_MsgHandler                        : FB_MSG_HANDLER;
  sL_MsgConfig                         : ST_MSG_CONFIG;
  fB_Msg                               : ARRAY [1..iC_NUM_MSG] OF FB_MESSAGE;
END_VAR

VAR PERSISTENT
  fI_PositionCappingClean              : REAL;           (*[mm]*)
  fI_PositionPark                      : REAL;           (*[mm]*)
  fI_PositionTolerance                 : REAL := 0.001;  (*[m]*)
  sI_SpeedDef                          : ST_SPEEDS;  (*Speed defs [mm/s]*)
END_VAR

VAR CONSTANT
  iC_NUM_MSG                           : INT  := 1;
END_VAR

//Limit switches for internal use
bL_ReferenceSensor := NOT bI_ReferenceSensor;

(*----------------------------------------------------------------------------------------------------------------------------------------------- *)
(*Running Conditions for Cleaning Unit  *)
(*----------------------------------------------------------------------------------------------------------------------------------------------- *)
IF I_MachineStatus.pSafetyOk AND I_MachineStatus.pMachineReady AND (wL_ErrorCode = 0 OR wL_ErrorCode.5)THEN  (*Dont check limit switch here*)
  bL_SafeRunningCondition := TRUE;
ELSE
  bL_SafeRunningCondition := FALSE;
END_IF;

bL_SafeMoveNeg := bL_SafeRunningCondition AND NOT bL_ReferenceSensor AND bI_SafeToMove;
bL_SafeMovePos := bL_SafeRunningCondition AND bI_SafeToMove;

(*Because the WcState sets an error for on cycle, we use this timer to check if the bus is down.*)
fb_TonDeviceOnline(IN := bI_DeviceOnline, PT := T#20MS);
fb_RTrigDeviceReset(CLK := bIDp_DeviceReset);
IF fb_TonDeviceOnline.Q OR fb_RTrigDeviceReset.Q THEN
  bL_RefKnown    := FALSE;        (*Reset Reference when link to device is lost, e.g. when machine power off*)
	wL_ErrorCode.9 := TRUE;
END_IF;

(*----------------------------------------------------------------------------------------------------------------------------------------------- *)
(*Position detection*)
(*----------------------------------------------------------------------------------------------------------------------------------------------- *)
IF     fB_Axis.fO_ActualPosition >= ((fI_PositionCappingClean / 1000) - fI_PositionTolerance)
   AND fB_Axis.fO_ActualPosition <= ((fI_PositionCappingClean / 1000) + fI_PositionTolerance)
THEN
  bL_InPosCappClean := TRUE;
  bL_InPosPark      := FALSE;
ELSIF  fB_Axis.fO_ActualPosition >= ((fI_PositionPark / 1000) - fI_PositionTolerance)
   AND fB_Axis.fO_ActualPosition <= ((fI_PositionPark / 1000) + fI_PositionTolerance)
THEN
  bL_InPosCappClean := FALSE;
  bL_InPosPark      := TRUE;
ELSE
  bL_InPosCappClean := FALSE;
  bL_InPosPark      := FALSE;
END_IF;


(*----------------------------------------------------------------------------------------------------------------------------------------------- *)
(* Axis control  *)
(*----------------------------------------------------------------------------------------------------------------------------------------------- *)
fB_Axis.bI_RegActive := bL_SafeRunningCondition AND NOT bL_Error; //Activate controller
fB_Axis.bI_EStop     := I_MachineStatus.pSafetyOk;                //negative logic for bI_EStop

fB_Axis(wI_StatusWord := wI_StatusWord ,lI_EncoderValue := lI_EncoderValue);

fB_Axis.bI_FaultReset := FALSE;

wO_ControlWord    := fB_Axis.wO_ControlWord;
iO_TargetVelocity := fB_Axis.iO_TargetVelocity;


(*----------------------------------------------------------------------------------------------------------------------------------------------- *)
(*Manuell move in hand mode (NOT bI_UsrAutoMode)*)
(*----------------------------------------------------------------------------------------------------------------------------------------------- *)
fb_RFTrigManualMove(CLK := sADS_CleanAxis.bI_ManualMove);
IF     NOT bI_UsrAutoMode 
   AND bI_UsrService
   AND bI_SafetyOk
   AND NOT bI_WatchdogError
THEN
  sADS_CleanAxis.setFeedback( bManualMoveCanEx := TRUE
                            , bManualMovekExec := sADS_CleanAxis.bO_ManualMovekExec        // do not change
                            , fAxisPositionVal := sADS_CleanAxis.sO_AxisPosition.fO_Val    // do not change
                            , wErrorCode       := sADS_CleanAxis.wO_ErrorCode              // do not change
                            , bBusy            := sADS_CleanAxis.bO_Busy                   // do not change
                            , bReady           := sADS_CleanAxis.bO_Ready                  // do not change
                            , bError           := sADS_CleanAxis.bO_Error                  // do not change
                            );

  IF sADS_CleanAxis.bI_ManualMove OR fb_RFTrigManualMove.FT THEN
    mManuellMove( bI_Do                  := sADS_CleanAxis.bI_ManualMove
                , fI_TargetPosition      := SEL( sADS_CleanAxis.bI_ManualMove
                                               , (fB_Axis.fO_ActualPosition * 1000)
                                               , sADS_CleanAxis.fI_ManualTargetPos)
                , fL_ManualMoveTolerance := fB_Axis.fI_Tolerance);
  END_IF
ELSE
  sADS_CleanAxis.setFeedback( bManualMoveCanEx := FALSE
                            , bManualMovekExec := sADS_CleanAxis.bO_ManualMovekExec        // do not change
                            , fAxisPositionVal := sADS_CleanAxis.sO_AxisPosition.fO_Val    // do not change
                            , wErrorCode       := sADS_CleanAxis.wO_ErrorCode              // do not change
                            , bBusy            := sADS_CleanAxis.bO_Busy                   // do not change
                            , bReady           := sADS_CleanAxis.bO_Ready                  // do not change
                            , bError           := sADS_CleanAxis.bO_Error                  // do not change
                            );
  sADS_CleanAxis.ResetCommands();

  IF fb_RFTrigManualMove.FT THEN
    mManuellMove( bI_Do                  := FALSE
                , fI_TargetPosition      := (fB_Axis.fO_ActualPosition * 1000)
                , fL_ManualMoveTolerance := fB_Axis.fI_Tolerance);
  END_IF
END_IF
(*Rest command if move is done*)
IF bL_Ready OR bL_Error THEN
  sADS_CleanAxis.ResetCommands();
END_IF

sL_CleanDevStatus := sStatus;

(*ADS Feedback*)
sADS_CleanAxis.setFeedback( bManualMoveCanEx := sADS_CleanAxis.bO_ManualMoveCanEx        // do not change
                          , bManualMovekExec := sADS_CleanAxis.bO_ManualMovekExec        // do not change
                          , fAxisPositionVal := fB_Axis.fO_ActualPosition * 1000
                          , wErrorCode       := wL_ErrorCode
                          , bBusy            := sL_CleanDevStatus.bBusy
                          , bReady           := sL_CleanDevStatus.bReady
                          , bError           := sL_CleanDevStatus.bError
                          );


(*----------------------------------------------------------------------------------------------------------------------------------------------- *)
(* Supervision  *)
(*----------------------------------------------------------------------------------------------------------------------------------------------- *)
(*
TODO: Supervisor
tL_TimerSurv.PT := T#3S;
tL_TimerSurv();
tL_TimerSensor.PT := T#105s  ;  (* 1meter at 10mm*)
tL_TimerSensor();*)

IF bL_FirstRun THEN
  bL_FirstRun     := FALSE;
  bL_memRefSensor := bL_ReferenceSensor;
END_IF;

(*----------------------------------------------------------------------------------------------------------------------- *)
(*--------------------------------- Fault Diagnosis and Management  ----------------------------------------------------- *)
(*----------------------------------------------------------------------------------------------------------------------- *)
mErrorHandling();

(*----------------------------------------------------------------------------------------------------------------------- *)
(* Messaging                                                                                                              *)
(*----------------------------------------------------------------------------------------------------------------------- *)
fB_MsgHandler();
fB_Msg[1](bI_Status := bL_Error);
fB_MsgQueue();

METHOD mAckError 
VAR_INPUT
END_VAR
wL_ErrorCode := 0;
mErrorHandling();
fB_Axis.bI_FaultReset := TRUE;
END_METHOD

METHOD mCapping : BOOL
VAR_INPUT
  iI_Step    : INT;
  bI_ExitCap : BOOL;
END_VAR
//Abort: Stop whereever axis is and return
IF bL_AbortReq THEN
  fB_Axis.bI_MoveEnable := FALSE;
  bL_Busy  := FALSE;
  bL_Ready := TRUE;

  RETURN;
END_IF

//Normal operation
bL_Ready := FALSE;
CASE iI_Step OF
	0: //Init - Check if axis is not activated, restore safety
    fB_Axis.bI_MoveEnable := FALSE;
		bL_Busy := FALSE;

  1: //Wait for PU axis to lift
    fB_Axis.bI_MoveEnable   := FALSE;
    bL_Busy                 := FALSE;
    
  2: //Wait for CU axis to move in
    mAckError();
    fB_Axis.fI_TargetPosition := (fI_PositionCappingClean / 1000);
    fB_Axis.fI_SpeedLimit     := sI_SpeedDef.fP_PlaceSpeed / 1000;
    
    IF bL_InPosCappClean THEN
      fB_Axis.bI_MoveEnable := FALSE;
      bL_Busy               := FALSE;
      bL_Ready              := TRUE;  //Operation complete
    ELSE
      fB_Axis.bI_MoveEnable := bL_SafeMovePos;
      bL_Busy               := TRUE;
    END_IF
    
  3: //Move CH to park positiom 
    fB_Axis.bI_MoveEnable   := FALSE;
    bL_Busy                 := FALSE;
    
  4: //Wait for PU axis to lower
    fB_Axis.bI_MoveEnable   := FALSE;
    bL_Busy                 := FALSE;
    
	5: //End - Do nothing, capping process active
    mAckError();
		bL_Busy  := FALSE;
    bL_Ready := TRUE;  //Operation complete

	ELSE
		bL_Busy  := FALSE;		
    bL_Ready := TRUE;  //Operation complete
END_CASE
END_METHOD

METHOD mCleaning : BOOL
VAR_INPUT
  iI_Step : INT;
END_VAR
//Abort: Stop whereever axis is and return
IF bL_AbortReq THEN
  fB_Axis.bI_MoveEnable := FALSE;
  bL_Busy  := FALSE;
  bL_Ready := TRUE;

  RETURN;
END_IF

//Normal operation
bL_Ready := FALSE;
CASE iI_Step OF
  0: //Init - Check if axis is not activated, restore safety
    bL_Busy := FALSE;

  1: //Wait for PU axis to lift
    fB_Axis.bI_MoveEnable   := FALSE;
    bL_Busy                 := FALSE;
    
  2: //Wait for CU axis to move in
    mAckError();
    fB_Axis.fI_TargetPosition := (fI_PositionCappingClean / 1000);
    fB_Axis.fI_SpeedLimit     := sI_SpeedDef.fP_PlaceSpeed / 1000;
    
    IF bL_InPosCappClean THEN
      fB_Axis.bI_MoveEnable := FALSE;
      bL_Busy               := FALSE;
      bL_Ready              := TRUE;  //Operation complete
    ELSE
      fB_Axis.bI_MoveEnable := bL_SafeMovePos;
      bL_Busy               := TRUE;
    END_IF
    
  3: //Wait for PU axis to lower
    fB_Axis.bI_MoveEnable   := FALSE;
    bL_Busy                 := FALSE;
    
  4: //Ensure CH axis is at starting position
    fB_Axis.bI_MoveEnable   := FALSE;
    bL_Busy                 := FALSE;
    
  5: //Move CH to clean start position
    fB_Axis.bI_MoveEnable   := FALSE;
    bL_Busy                 := FALSE;

  6: //Wait until cleaning equipment ready
    fB_Axis.bI_MoveEnable   := FALSE;
    bL_Busy                 := FALSE;
    
  7: //Cleaning
    fB_Axis.bI_MoveEnable   := FALSE;
    bL_Busy                 := FALSE;  
    
  8: //Wait until cleaning equipment ready
    fB_Axis.bI_MoveEnable   := FALSE;
    bL_Busy                 := FALSE;
    
  9: //Move CH to end position
    fB_Axis.bI_MoveEnable   := FALSE;
    bL_Busy                 := FALSE;  
    
  10: //Wait for PU axis to lift
    fB_Axis.bI_MoveEnable   := FALSE;
    bL_Busy                 := FALSE;  
  
  11: //Move CH back to start 
    fB_Axis.bI_MoveEnable   := FALSE;
    bL_Busy                 := FALSE;  

  12: //Wait for PU axis to lower
    fB_Axis.bI_MoveEnable   := FALSE;
    bL_Busy                 := FALSE;
    
  13: //End
    fB_Axis.bI_MoveEnable   := FALSE;
    bL_Busy                 := FALSE;  
    bL_Ready                := TRUE;  //Operation complete

  ELSE
    bL_Busy  := FALSE;    
    bL_Ready := TRUE;  //Operation complete
END_CASE
END_METHOD

METHOD PRIVATE mErrorHandling
VAR_INPUT
END_VAR
fB_Msg[1].bI_Status := FALSE;

IF (sI_SpeedDef.fP_PlaceSpeed = 0) OR (sI_SpeedDef.fP_WorkSpeed = 0) OR (sI_SpeedDef.fP_ServiceSpeed = 0) THEN	(* Speed Configuration not done *)
	wL_ErrorCode.6 := TRUE;
END_IF;

IF (fI_PositionCappingClean = 0) THEN		(* Position Configuration not done *)
	wL_ErrorCode.7 := TRUE;
END_IF;

IF fB_Axis.eO_EL7201Status = eFault  THEN
	wL_ErrorCode.8 := TRUE;						(* EL7342 module fault *)
	fB_Msg[1].bI_Status := TRUE;
END_IF;


IF wl_ErrorCode = 0 THEN
	bL_Error := FALSE;
ELSE
	bL_Error := TRUE;
END_IF;
END_METHOD

METHOD mErrorRecovery : BOOL
VAR_INPUT
    iI_Step : INT;
END_VAR
//Do nothing
bL_Busy  := FALSE;
bL_Ready := TRUE;
END_METHOD

METHOD mInit
VAR_INPUT
END_VAR
(*Messages*)
sL_MsgConfig.bI_Enable       := TRUE;
sL_MsgConfig.pI_FbMsgHandler := ADR(fB_MsgHandler);
fB_MsgHandler.pI_MsgQueue    := ADR(fB_MsgQueue);
fB_MsgQueue.pI_MsgInterface  := ADR(sADS_CleanAxis.sO_Message);
fB_MsgQueue.cI_MaxElement    := 5;

fB_Msg[1].iI_MsgLocation     := TO_INT(eMa_BLK_CLEANAXIS);
fB_Msg[1].pI_MsgConfig       := ADR(sL_MsgConfig);
fB_Msg[1].iI_MsgNumber       := eCMa_AxisErrorX;
END_METHOD

METHOD mManuellMove : BOOL
VAR_INPUT
  bI_Do                  : BOOL;
  fI_TargetPosition      : REAL;
  fL_ManualMoveTolerance : REAL;
END_VAR
fB_Axis.fI_SpeedLimit     := sI_SpeedDef.fP_ServiceSpeed / 1000;
fB_Axis.fI_TargetPosition := fI_TargetPosition / 1000;
IF fB_Axis.fI_TargetPosition > fB_Axis.fO_ActualPosition THEN
  fB_Axis.bI_MoveEnable   := bI_Do AND bL_SafeMovePos;
ELSIF fB_Axis.fI_TargetPosition < fB_Axis.fO_ActualPosition THEN
  fB_Axis.bI_MoveEnable   := bI_Do AND bL_SafeMoveNeg;
ELSE
  fB_Axis.bI_MoveEnable   := bI_Do;
END_IF

bL_Busy  := ABS(fB_Axis.fI_TargetPosition - fB_Axis.fO_ActualPosition) > fL_ManualMoveTolerance;
bL_Ready := NOT (ABS(fB_Axis.fI_TargetPosition - fB_Axis.fO_ActualPosition) > fL_ManualMoveTolerance);  //Operation complete
END_METHOD

METHOD mProduction : BOOL
VAR_INPUT
  iI_Step : INT;
END_VAR
//Abort: Stop whereever axis is and return
IF bL_AbortReq THEN
  fB_Axis.bI_MoveEnable := FALSE;
  bL_Busy  := FALSE;
  bL_Ready := TRUE;

  RETURN;
END_IF

//Normal operation
bL_Ready := FALSE;
CASE iI_Step OF
  0: //Init - Check if axis is not activated, restore safety
    bL_Busy := FALSE;

  1: //Wait for PU axis to lift
    fB_Axis.bI_MoveEnable   := FALSE;
    bL_Busy                 := FALSE;
    
  2: //Wait for CU axis to move out
    mAckError();
    fB_Axis.fI_TargetPosition := (fI_PositionPark / 1000);
    fB_Axis.fI_SpeedLimit     := sI_SpeedDef.fP_PlaceSpeed / 1000;
    
    IF bL_InPosPark THEN
      fB_Axis.bI_MoveEnable := FALSE;
      bL_Busy               := FALSE;
      bL_Ready              := TRUE;  //Operation complete
    ELSE
      fB_Axis.bI_MoveEnable := bL_SafeMoveNeg;
      bL_Busy               := TRUE;
    END_IF
    
  3: //Wait for PU axis to lower
    fB_Axis.bI_MoveEnable   := FALSE;
    bL_Busy                 := FALSE;
    
  4: //End
    fB_Axis.bI_MoveEnable := FALSE;
    bL_Busy               := FALSE;  
    bL_Ready              := TRUE;  //Operation complete

  ELSE
    bL_Busy  := FALSE;    
    bL_Ready := TRUE;  //Operation complete
END_CASE
END_METHOD

METHOD mService : BOOL
VAR_INPUT
  iI_Step : INT;
END_VAR
//Abort: Stop whereever axis is and return
IF bL_AbortReq THEN
  fB_Axis.bI_MoveEnable := FALSE;
  bL_Busy  := FALSE;
  bL_Ready := TRUE;

  RETURN;
END_IF

//Normal operation
bL_Ready := FALSE;
CASE iI_Step OF
  0: //Init - Check if axis is not activated, restore safety
    bL_Busy := FALSE;

  1: //Wait for PU axis to lift to ExitCapping
    fB_Axis.bI_MoveEnable   := FALSE;
    bL_Busy                 := FALSE;
    
  2: //Wait for CU axis to move in
    mAckError();
    fB_Axis.fI_TargetPosition := (fI_PositionPark / 1000);
    fB_Axis.fI_SpeedLimit     := sI_SpeedDef.fP_PlaceSpeed / 1000;
    
    IF bL_InPosPark THEN
      fB_Axis.bI_MoveEnable := FALSE;
      bL_Busy               := FALSE;
      bL_Ready              := TRUE;  //Operation complete
    ELSE
      fB_Axis.bI_MoveEnable := bL_SafeMoveNeg;
      bL_Busy               := TRUE;
    END_IF
    
  3: //End
    fB_Axis.bI_MoveEnable := FALSE;
    bL_Busy               := FALSE;  
    bL_Ready              := TRUE;

  ELSE
    bL_Busy  := FALSE;    
    bL_Ready := TRUE;  //Operation complete
END_CASE
END_METHOD

METHOD mStartup : BOOL
VAR_INPUT
  iI_Step : INT;
END_VAR
CASE iI_Step OF
	0: //Init - Check if axis is not activated, restore safety
		bL_Busy := FALSE;

	1: //Wait until other axes in place
		bL_Busy := FALSE;

	2: //Begin - Init CU axis if NOT bL_RefKnown
    bL_Busy  := NOT bL_RefKnown;
    bL_Ready := bL_RefKnown;
    
    fB_Axis.bI_SetPosition := bL_RefKnown;
    
    IF NOT bL_RefKnown THEN  (* if the CU axis hasn't been initialized with Ref Sensor*)
      IF bL_ReferenceSensor AND NOT bL_memRefSensor AND NOT bL_RefKnown THEN
        bL_RefKnown             := TRUE;                      (* When the sensor is activated, Save the correction value*)
        fB_Axis.bI_SetPosition  := TRUE;                      (*Initialize position to preset value*)
        fB_Axis.bI_MoveEnable   := FALSE;
        bL_Ready                := TRUE;
      ELSE
        IF bL_ReferenceSensor AND bL_memRefSensor THEN
          fB_Axis.fI_TargetPosition := fB_Axis.fO_ActualPosition + 0.01;  (*@@@@CONST, change to JOG_NEGATIVE*)
          fB_Axis.fI_SpeedLimit     := sI_SpeedDef.fP_ServiceSpeed / 1000;     (* Start backward motion, the motor will run until Ref Sensor is ON*)
          fB_Axis.bI_MoveEnable     := bL_SafeMovePos;
        ELSE
          fB_Axis.fI_TargetPosition := -100.0;                               (*@@@@CONST, change to JOG_NEGATIVE*)
          fB_Axis.fI_SpeedLimit     := sI_SpeedDef.fP_ServiceSpeed / 1000;  (* Start backward motion, the motor will run until Ref Sensor is ON*)
          fB_Axis.bI_MoveEnable     := bL_SafeMoveNeg;
        END_IF;
      END_IF;
    END_IF;

    bL_memRefSensor := bL_ReferenceSensor;				(* Memorization of the Ref sensor state for edge detection*)

	3,4: //End
		bL_Busy  := FALSE;		
    bL_Ready := TRUE;  //Operation complete

	ELSE
		bL_Busy  := FALSE;		
    bL_Ready := TRUE;  //Operation complete
END_CASE
END_METHOD

{attribute 'monitoring' := 'call'}
PROPERTY pInPosCappingClean : BOOL
GET
pInPosCappingClean := bL_InPosCappClean;
END_GET
END_PROPERTY

{attribute 'monitoring' := 'call'}
PROPERTY pInPosPark : bool
GET
pInPosPark := bL_InPosPark;
END_GET
END_PROPERTY

END_FUNCTION_BLOCK

// ---- POUs/Machine/CleaningStation/FB_CleaningMotorAxisPU.TcPOU
FUNCTION_BLOCK FB_CleaningMotorAxisPU EXTENDS FB_CleanDevice
VAR_INPUT
  bI_SafeToMove                        : BOOL;
  bI_Emergency                         : BOOL;
  bI_WatchdogError                     : BOOL;
  bI_SafetyOk                          : BOOL;
  bI_MachineReady                      : BOOL;
  bI_UsrAutoMode                       : BOOL;
  bI_UsrService                        : BOOL;
  bI_DevOpActive                       : BOOL;
	fI_SheetThickness                    : REAL := 0.000; (*Sheet thickness (Production Mode) [mm]*)
  
  //Limit switches
  bI_SensorTop                  AT %I* : BOOL;  (*Physical sensor feedback for top position*)
  bI_SensorBottom               AT %I* : BOOL;  (*Physical sensor feedback for bottom position*)
  
  //Inputs from EL7201 Terminal
  wI_StatusWord                 AT %I* : UINT; (*Status word: 6041:0*)
  lI_EncoderValue               AT %I* : DINT; (*Encoder value*)
  bI_DeviceOnline               AT %I* : BOOL; (*Check link to device*)
  
  fB_Axis                              : FB_EL7201;    //Axis controller
END_VAR

VAR_OUTPUT
  //Outputs to EL7201 Terminal
  wO_ControlWord                AT %Q* : UINT;                         (*Control word:  6040:0*)
  iO_TargetVelocity             AT %Q* : DINT;                         (*Target velocity:  60FF:0*)
END_VAR

VAR
  sADS_CleanAxis                       : FB_ADS_CleanAxis;     //ST_ADS_CLEAN_AXIS;

  fb_TonDeviceOnline                   : TON;
	bIDp_DeviceReset                     : BOOL := FALSE;
	fb_RTrigDeviceReset                  : R_TRIG;
  fb_RFTrigPrintEnabled                : RF_TRIG;

  bL_DriveToWaitPos                    : BOOL;
  bL_DriveToPrintPos                   : BOOL;

  bL_SafeRunningCondition              : BOOL;
  bL_SafeMoveNeg                       : BOOL;
  bL_SafeMovePos                       : BOOL;
  bL_FirstRun                          : BOOL := TRUE;

  fL_PrintPosition                     : REAL;  (*[m]*)
  fL_PrintPositionMM                   : REAL;  (*[mm]*)
  bL_InPosService                      : BOOL;
  bL_InPosClean1                       : BOOL;
  bL_InPosClean2                       : BOOL;
  bL_InPosWait                         : BOOL;
  bL_InPosPrint                        : BOOL;
  bL_HigherPosWait                     : BOOL;
  bL_HigherPosC1                       : BOOL;
  
  fb_RFTrigManualMove                  : RF_TRIG;
  sL_CleanDevStatus                    : ST_CLEANING_DEV_STATUS;

  bL_MemSensorTop                      : BOOL;
  bL_MemSensorBottom                   : BOOL;

  wL_ErrorCode                         : WORD;
  
  (*Messaging*)
  fB_MsgQueue                          : FB_MSG_QUEUE;
  fB_MsgHandler                        : FB_MSG_HANDLER;
  sL_MsgConfig                         : ST_MSG_CONFIG;
  fB_Msg                               : ARRAY [1..iC_NUM_MSG] OF FB_MESSAGE;
END_VAR

VAR PERSISTENT
  fI_PositionService                   : REAL;  (*[mm]*)
  fI_PositionWait                      : REAL;  (*[mm]*)
  fI_PositionClean1                    : REAL;  (*[mm]*)
  fI_PositionClean2                    : REAL;  (*[mm]*)
  fI_PositionPrint                     : REAL;  (*[mm]*)
  fL_SetPositionValue                  : REAL := 10.2;    (*[mm]*)
  fI_PositionTolerance                 : REAL := 0.0001;  (*[m]*)
  fI_PositionTolerance2                : REAL := 0.005;   (*[m]*)
  sI_SpeedDef                          : ST_SPEEDS;  (*Speed defs [mm/s]*)
END_VAR

VAR CONSTANT
  iC_NUM_MSG                           : INT  := 1;
END_VAR

(*----------------------------------------------------------------------------------------------------------------------------------------------- *)
(*Running Conditions for Cleaning Head  *)
(*----------------------------------------------------------------------------------------------------------------------------------------------- *)
IF I_MachineStatus.pSafetyOk AND I_MachineStatus.pMachineReady AND (wL_ErrorCode = 0 OR wL_ErrorCode.5)THEN  (*Dont check limit switch here*)
  bL_SafeRunningCondition := TRUE;
ELSE
  bL_SafeRunningCondition := FALSE;
END_IF;

bL_SafeMoveNeg := bL_SafeRunningCondition AND bI_SensorBottom AND bI_SafeToMove;
bL_SafeMovePos := bL_SafeRunningCondition AND bI_SensorTop;

(*Because the WcState sets an error for on cycle, we use this timer to check if the bus is down.*)
fb_TonDeviceOnline(IN := bI_DeviceOnline, PT := T#20MS);
fb_RTrigDeviceReset(CLK := bIDp_DeviceReset);
IF fb_TonDeviceOnline.Q OR fb_RTrigDeviceReset.Q THEN
  bL_RefKnown    := FALSE;        (*Reset Reference when link to device is lost, e.g. when machine power off*)
	wL_ErrorCode.9 := TRUE;
END_IF;

(*----------------------------------------------------------------------------------------------------------------------------------------------- *)
(*Position detection*)
(*----------------------------------------------------------------------------------------------------------------------------------------------- *)
fL_PrintPositionMM := fI_PositionPrint + fI_SheetThickness;
fL_PrintPosition   := (fL_PrintPositionMM / 1000);

IF     fB_Axis.fO_ActualPosition >= ((fI_PositionWait / 1000) - (fI_PositionTolerance / 1000))
   AND fB_Axis.fO_ActualPosition <= ((fI_PositionWait / 1000) + (fI_PositionTolerance / 1000))
THEN
  bL_InPosService := FALSE;
  bL_InPosClean1  := FALSE;
  bL_InPosClean2  := FALSE;
  bL_InPosWait    := TRUE;
  bL_InPosPrint   := FALSE;
ELSIF  fB_Axis.fO_ActualPosition >= (fL_PrintPosition - fI_PositionTolerance)
   AND fB_Axis.fO_ActualPosition <= (fL_PrintPosition + fI_PositionTolerance)
THEN
  bL_InPosService := FALSE;
  bL_InPosClean1  := FALSE;
  bL_InPosClean2  := FALSE;
  bL_InPosWait    := FALSE;
  bL_InPosPrint   := TRUE;
ELSIF  fB_Axis.fO_ActualPosition >= ((fI_PositionService / 1000) - fI_PositionTolerance)
   AND fB_Axis.fO_ActualPosition <= ((fI_PositionService / 1000) + fI_PositionTolerance)
THEN
  bL_InPosService := TRUE;
  bL_InPosClean1  := FALSE;
  bL_InPosClean2  := FALSE;
  bL_InPosWait    := FALSE;
  bL_InPosPrint   := FALSE;
ELSIF  fB_Axis.fO_ActualPosition >= ((fI_PositionClean1 / 1000) - fI_PositionTolerance)
   AND fB_Axis.fO_ActualPosition <= ((fI_PositionClean1 / 1000) + fI_PositionTolerance)
THEN
  bL_InPosService := FALSE;
  bL_InPosClean1  := TRUE;
  IF fI_PositionClean1 = fI_PositionClean2 THEN
    bL_InPosClean2  := TRUE;
  ELSE
    bL_InPosClean2  := FALSE;
	END_IF
  bL_InPosWait    := FALSE;
  bL_InPosPrint   := FALSE;
ELSIF  fB_Axis.fO_ActualPosition >= ((fI_PositionClean2 / 1000) - fI_PositionTolerance)
   AND fB_Axis.fO_ActualPosition <= ((fI_PositionClean2 / 1000) + fI_PositionTolerance)
THEN
  bL_InPosService := FALSE;
  bL_InPosClean1  := FALSE;
  bL_InPosClean2  := TRUE;
  bL_InPosWait    := FALSE;
  bL_InPosPrint   := FALSE;
ELSE
  bL_InPosService := FALSE;
  bL_InPosClean1  := FALSE;
  bL_InPosClean2  := FALSE;
  bL_InPosWait    := FALSE;
  bL_InPosPrint   := FALSE;
END_IF;
bL_HigherPosWait := fB_Axis.fO_ActualPosition >= ((fI_PositionWait   / 1000) + fI_PositionTolerance2);
bL_HigherPosC1   := fB_Axis.fO_ActualPosition >= ((fI_PositionClean1 / 1000));

(*----------------------------------------------------------------------------------------------------------------------------------------------- *)
(* Axis control  *)
(*----------------------------------------------------------------------------------------------------------------------------------------------- *)
fB_Axis.bI_RegActive        := bL_SafeRunningCondition AND NOT bL_Error; //Activate controller
fB_Axis.bI_EStop            := I_MachineStatus.pSafetyOk;                //negative logic for bI_EStop
fB_Axis.fI_SetPositionValue := fL_SetPositionValue / 1000;

fB_Axis(wI_StatusWord := wI_StatusWord ,lI_EncoderValue := lI_EncoderValue);

fB_Axis.bI_FaultReset := FALSE;

wO_ControlWord    := fB_Axis.wO_ControlWord;
iO_TargetVelocity := fB_Axis.iO_TargetVelocity;

IF fB_Axis.fL_OffsetEncoder > 0 THEN
	bL_RefKnown := TRUE;
ELSE
	bL_RefKnown := FALSE;
END_IF;


(*----------------------------------------------------------------------------------------------------------------------------------------------- *)
(*Manuell move in hand mode (NOT bI_UsrAutoMode)*)
(*----------------------------------------------------------------------------------------------------------------------------------------------- *)
fb_RFTrigManualMove(CLK := sADS_CleanAxis.bI_ManualMove);
IF     NOT bI_UsrAutoMode 
   AND bI_UsrService
   AND bI_SafetyOk
   AND NOT bI_WatchdogError
THEN
  sADS_CleanAxis.setFeedback( bManualMoveCanEx := TRUE
                            , bManualMovekExec := sADS_CleanAxis.bO_ManualMovekExec        // do not change
                            , fAxisPositionVal := sADS_CleanAxis.sO_AxisPosition.fO_Val    // do not change
                            , wErrorCode       := sADS_CleanAxis.wO_ErrorCode              // do not change
                            , bBusy            := sADS_CleanAxis.bO_Busy                   // do not change
                            , bReady           := sADS_CleanAxis.bO_Ready                  // do not change
                            , bError           := sADS_CleanAxis.bO_Error                  // do not change
                            );

  IF sADS_CleanAxis.bI_ManualMove OR fb_RFTrigManualMove.FT THEN
    mManuellMove( bI_Do                  := sADS_CleanAxis.bI_ManualMove
                , fI_TargetPosition      := SEL( sADS_CleanAxis.bI_ManualMove
                                               , (fB_Axis.fO_ActualPosition * 1000)
                                               , sADS_CleanAxis.fI_ManualTargetPos)
                , fL_ManualMoveTolerance := fB_Axis.fI_Tolerance);
  END_IF
ELSE
  sADS_CleanAxis.setFeedback( bManualMoveCanEx := FALSE
                            , bManualMovekExec := sADS_CleanAxis.bO_ManualMovekExec        // do not change
                            , fAxisPositionVal := sADS_CleanAxis.sO_AxisPosition.fO_Val    // do not change
                            , wErrorCode       := sADS_CleanAxis.wO_ErrorCode              // do not change
                            , bBusy            := sADS_CleanAxis.bO_Busy                   // do not change
                            , bReady           := sADS_CleanAxis.bO_Ready                  // do not change
                            , bError           := sADS_CleanAxis.bO_Error                  // do not change
                            );
  sADS_CleanAxis.ResetCommands();

